LIN {X 0,Y 181.247,Z 724.094,A -85,B 0,C 180,E1 25006.197,E2 25006.197} C_VEL
LIN {X 0,Y 212.827,Z 697.919,A -85,B 0,C 180,E1 25010.796,E2 25010.796} C_VEL
LIN {X 0,Y 227.243,Z 683.519,A -85,B 0,C 180,E1 25012.44,E2 25012.44} C_VEL
LIN {X 0,Y 228.905,Z 680.992,A -85,B 0,C 180,E1 25016.21,E2 25016.21} C_VEL
LIN {X 0,Y 228.998,Z 681.06,A -85,B 0,C 180,E1 25020.002,E2 25020.002} C_VEL
LIN {X 0,Y 227.551,Z 683.584,A -85,B 0,C 180,E1 25023.524,E2 25023.524} C_VEL
LIN {X 0,Y 198.346,Z 711.493,A -85,B 0,C 180,E1 25027.069,E2 25027.069} C_VEL
LIN {X 0,Y 166.945,Z 735.496,A -85,B 0,C 180,E1 25032.577,E2 25032.577} C_VEL
LIN {X 0,Y 134.271,Z 755.47,A -85,B 0,C 180,E1 25041.514,E2 25041.514} C_VEL
LIN {X 0,Y 104.1,Z 770.587,A -85,B 0,C 180,E1 25057.124,E2 25057.124} C_VEL
LIN {X 0,Y 86.325,Z 778.801,A -85,B 0,C 180,E1 25078.251,E2 25078.251} C_VEL
LIN {X 0,Y 80.671,Z 781.977,A -85,B 0,C 180,E1 25099.182,E2 25099.182} C_VEL
LIN {X 0,Y 80.808,Z 782.413,A -85,B 0,C 180,E1 25110,E2 25110} C_VEL
LIN {X 0,Y 83.389,Z 780.22,A -85,B 0,C 180,E1 25134.788,E2 25134.788} C_VEL
LIN {X 0,Y 97.45,Z 773.708,A -85,B 0,C 180,E1 25157.173,E2 25157.173} C_VEL
LIN {X 0,Y 123.333,Z 761.326,A -85,B 0,C 180,E1 25174.086,E2 25174.086} C_VEL
LIN {X 0,Y 156.668,Z 742.373,A -85,B 0,C 180,E1 25185.118,E2 25185.118} C_VEL
LIN {X 0,Y 191.224,Z 717.631,A -85,B 0,C 180,E1 25191.795,E2 25191.795} C_VEL
LIN {X 0,Y 222.942,Z 688.687,A -85,B 0,C 180,E1 25195.995,E2 25195.995} C_VEL
LIN {X 0,Y 227.55,Z 683.825,A -85,B 0,C 180,E1 25196.478,E2 25196.478} C_VEL
LIN {X 0,Y 229.058,Z 681.251,A -85,B 0,C 180,E1 25199.998,E2 25199.998} C_VEL
LIN {X 0,Y 228.87,Z 681.291,A -85,B 0,C 180,E1 25203.791,E2 25203.791} C_VEL
LIN {X 0,Y 227.892,Z 682.996,A -85,B 0,C 180,E1 25207.158,E2 25207.158} C_VEL
LIN {X 0,Y 219.93,Z 691.3,A -85,B 0,C 180,E1 25208.319,E2 25208.319} C_VEL
LIN {X 0,Y 189.42,Z 718.093,A -85,B 0,C 180,E1 25212.372,E2 25212.372} C_VEL
LIN {X 0,Y 157.043,Z 740.418,A -85,B 0,C 180,E1 25218.724,E2 25218.724} C_VEL
LIN {X 0,Y 125.362,Z 757.593,A -85,B 0,C 180,E1 25228.881,E2 25228.881} C_VEL
LIN {X 0,Y 98.281,Z 769.456,A -85,B 0,C 180,E1 25246.11,E2 25246.11} C_VEL
LIN {X 0,Y 83.688,Z 775.171,A -85,B 0,C 180,E1 25268.786,E2 25268.786} C_VEL
LIN {X 0,Y 81.015,Z 776.528,A -85,B 0,C 180,E1 25290,E2 25290} C_VEL
LIN {X 0,Y 83.704,Z 775.133,A -85,B 0,C 180,E1 25311.21,E2 25311.21} C_VEL
LIN {X 0,Y 98.34,Z 769.389,A -85,B 0,C 180,E1 25333.857,E2 25333.857} C_VEL
LIN {X 0,Y 126.011,Z 757.227,A -85,B 0,C 180,E1 25351.281,E2 25351.281} C_VEL
LIN {X 0,Y 148.843,Z 745.136,A -85,B 0,C 180,E1 25359.119,E2 25359.119} C_VEL
LIN {X 0,Y 159.683,Z 738.038,A -85,B 0,C 180,E1 25363.519,E2 25363.519} C_VEL
LIN {X 0,Y 171.008,Z 730.237,A -85,B 0,C 180,E1 25367.284,E2 25367.284} C_VEL
LIN {X 0,Y 202.656,Z 706.253,A -85,B 0,C 180,E1 25371.877,E2 25371.877} C_VEL
LIN {X 0,Y 222.664,Z 687.627,A -85,B 0,C 180,E1 25374.254,E2 25374.254} C_VEL
LIN {X 0,Y 223.276,Z 686.711,A -85,B 0,C 180,E1 25376.114,E2 25376.114} C_VEL
LIN {X 0,Y 222.89,Z 687.51,A -85,B 0,C 180,E1 25381.189,E2 25381.189} C_VEL
LIN {X 0,Y 221.964,Z 688.666,A -85,B 0,C 180,E1 25381.969,E2 25381.969} C_VEL
LIN {X 0,Y 190.199,Z 717.114,A -85,B 0,C 180,E1 25385.675,E2 25385.675} C_VEL
LIN {X 0,Y 154.741,Z 741.948,A -85,B 0,C 180,E1 25391.903,E2 25391.903} C_VEL
LIN {X 0,Y 120.508,Z 760.698,A -85,B 0,C 180,E1 25402.146,E2 25402.146} C_VEL
LIN {X 0,Y 90.513,Z 773.971,A -85,B 0,C 180,E1 25420.57,E2 25420.57} C_VEL
LIN {X 0,Y 75.014,Z 780.476,A -85,B 0,C 180,E1 25446.19,E2 25446.19} C_VEL
LIN {X 0,Y 72.87,Z 782.124,A -85,B 0,C 180,E1 25470,E2 25470} C_VEL
LIN {X 0,Y 75.013,Z 780.5,A -85,B 0,C 180,E1 25493.809,E2 25493.809} C_VEL
LIN {X 0,Y 90.48,Z 774.015,A -85,B 0,C 180,E1 25519.441,E2 25519.441} C_VEL
LIN {X 0,Y 120.494,Z 760.781,A -85,B 0,C 180,E1 25537.852,E2 25537.852} C_VEL
LIN {X 0,Y 154.748,Z 742.066,A -85,B 0,C 180,E1 25548.084,E2 25548.084} C_VEL
LIN {X 0,Y 190.221,Z 717.304,A -85,B 0,C 180,E1 25554.259,E2 25554.259} C_VEL
LIN {X 0,Y 222.009,Z 688.863,A -85,B 0,C 180,E1 25558.04,E2 25558.04} C_VEL
LIN {X 0,Y 223.412,Z 686.977,A -85,B 0,C 180,E1 25559.998,E2 25559.998} C_VEL
LIN {X 0,Y 222.855,Z 687.56,A -85,B 0,C 180,E1 25565.044,E2 25565.044} C_VEL
LIN {X 0,Y 222.649,Z 687.908,A -85,B 0,C 180,E1 25565.739,E2 25565.739} C_VEL
LIN {X 0,Y 190.138,Z 716.678,A -85,B 0,C 180,E1 25569.637,E2 25569.637} C_VEL
LIN {X 0,Y 157.034,Z 739.31,A -85,B 0,C 180,E1 25575.376,E2 25575.376} C_VEL
LIN {X 0,Y 121.669,Z 757.885,A -85,B 0,C 180,E1 25585.551,E2 25585.551} C_VEL
LIN {X 0,Y 92.636,Z 769.747,A -85,B 0,C 180,E1 25602.649,E2 25602.649} C_VEL
LIN {X 0,Y 76.32,Z 775.46,A -85,B 0,C 180,E1 25626.623,E2 25626.623} C_VEL
LIN {X 0,Y 73.116,Z 776.815,A -85,B 0,C 180,E1 25650,E2 25650} C_VEL
LIN {X 0,Y 76.336,Z 775.423,A -85,B 0,C 180,E1 25673.372,E2 25673.372} C_VEL
LIN {X 0,Y 92.69,Z 769.681,A -85,B 0,C 180,E1 25697.316,E2 25697.316} C_VEL
LIN {X 0,Y 122.329,Z 757.522,A -85,B 0,C 180,E1 25714.606,E2 25714.606} C_VEL
LIN {X 0,Y 157.068,Z 739.149,A -85,B 0,C 180,E1 25724.581,E2 25724.581} C_VEL
LIN {X 0,Y 171.008,Z 730.237,A -85,B 0,C 180,E1 25727.284,E2 25727.284} C_VEL
LIN {X 0,Y 182.635,Z 721.723,A -85,B 0,C 180,E1 25730.535,E2 25730.535} C_VEL
LIN {X 0,Y 192.75,Z 713.822,A -85,B 0,C 180,E1 25733.112,E2 25733.112} C_VEL
LIN {X 0,Y 194.377,Z 712.525,A -85,B 0,C 180,E1 25733.326,E2 25733.326} C_VEL
LIN {X 0,Y 216.534,Z 693.283,A -85,B 0,C 180,E1 25735.643,E2 25735.643} C_VEL
LIN {X 0,Y 217.51,Z 692.345,A -85,B 0,C 180,E1 25736.011,E2 25736.011} C_VEL
LIN {X 0,Y 217.609,Z 692.411,A -85,B 0,C 180,E1 25740.002,E2 25740.002} C_VEL
LIN {X 0,Y 202.192,Z 706.448,A -85,B 0,C 180,E1 25741.753,E2 25741.753} C_VEL
LIN {X 0,Y 169.875,Z 731.007,A -85,B 0,C 180,E1 25745.966,E2 25745.966} C_VEL
LIN {X 0,Y 135.641,Z 751.45,A -85,B 0,C 180,E1 25752.902,E2 25752.902} C_VEL
LIN {X 0,Y 103.811,Z 766.412,A -85,B 0,C 180,E1 25764.273,E2 25764.273} C_VEL
LIN {X 0,Y 76.451,Z 776.915,A -85,B 0,C 180,E1 25786.117,E2 25786.117} C_VEL
LIN {X 0,Y 67.715,Z 780.182,A -85,B 0,C 180,E1 25803.435,E2 25803.435} C_VEL
LIN {X 0,Y 64.928,Z 781.835,A -85,B 0,C 180,E1 25830,E2 25830} C_VEL
LIN {X 0,Y 67.715,Z 780.207,A -85,B 0,C 180,E1 25856.564,E2 25856.564} C_VEL
LIN {X 0,Y 84.983,Z 773.851,A -85,B 0,C 180,E1 25883.298,E2 25883.298} C_VEL
LIN {X 0,Y 115.267,Z 761.512,A -85,B 0,C 180,E1 25900.71,E2 25900.71} C_VEL
LIN {X 0,Y 149.728,Z 743.767,A -85,B 0,C 180,E1 25910.392,E2 25910.392} C_VEL
LIN {X 0,Y 184.033,Z 721.156,A -85,B 0,C 180,E1 25916.015,E2 25916.015} C_VEL
LIN {X 0,Y 215.219,Z 694.933,A -85,B 0,C 180,E1 25919.546,E2 25919.546} C_VEL
LIN {X 0,Y 217.661,Z 692.593,A -85,B 0,C 180,E1 25919.998,E2 25919.998} C_VEL
LIN {X 0,Y 217.464,Z 692.627,A -85,B 0,C 180,E1 25923.99,E2 25923.99} C_VEL
LIN {X 0,Y 205.321,Z 703.66,A -85,B 0,C 180,E1 25925.406,E2 25925.406} C_VEL
LIN {X 0,Y 174.486,Z 727.337,A -85,B 0,C 180,E1 25929.217,E2 25929.217} C_VEL
LIN {X 0,Y 141.335,Z 747.205,A -85,B 0,C 180,E1 25935.383,E2 25935.383} C_VEL
LIN {X 0,Y 106.184,Z 763.204,A -85,B 0,C 180,E1 25947.029,E2 25947.029} C_VEL
LIN {X 0,Y 78.516,Z 772.86,A -85,B 0,C 180,E1 25967.55,E2 25967.55} C_VEL
LIN {X 0,Y 65.738,Z 776.783,A -85,B 0,C 180,E1 25996.684,E2 25996.684} C_VEL
LIN {X 0,Y 65.199,Z 777.103,A -85,B 0,C 180,E1 26010,E2 26010} C_VEL
LIN {X 0,Y 69.067,Z 775.715,A -85,B 0,C 180,E1 26036.006,E2 26036.006} C_VEL
LIN {X 0,Y 87.414,Z 769.976,A -85,B 0,C 180,E1 26061.212,E2 26061.212} C_VEL
LIN {X 0,Y 118.16,Z 758.2,A -85,B 0,C 180,E1 26077.791,E2 26077.791} C_VEL
LIN {X 0,Y 151.659,Z 741.427,A -85,B 0,C 180,E1 26086.761,E2 26086.761} C_VEL
LIN {X 0,Y 186.136,Z 718.9,A -85,B 0,C 180,E1 26092.315,E2 26092.315} C_VEL
LIN {X 0,Y 194.377,Z 712.525,A -85,B 0,C 180,E1 26093.326,E2 26093.326} C_VEL
LIN {X 0,Y 201.791,Z 706.345,A -85,B 0,C 180,E1 26095.31,E2 26095.31} C_VEL
LIN {X 0,Y 209.229,Z 699.942,A -85,B 0,C 180,E1 26097.168,E2 26097.168} C_VEL
LIN {X 0,Y 211.637,Z 697.732,A -85,B 0,C 180,E1 26097.44,E2 26097.44} C_VEL
LIN {X 0,Y 211.653,Z 697.751,A -85,B 0,C 180,E1 26098.428,E2 26098.428} C_VEL
LIN {X 0,Y 178.493,Z 724.38,A -85,B 0,C 180,E1 26101.989,E2 26101.989} C_VEL
LIN {X 0,Y 141.371,Z 747.345,A -85,B 0,C 180,E1 26107.816,E2 26107.816} C_VEL
LIN {X 0,Y 103.874,Z 764.915,A -85,B 0,C 180,E1 26118.651,E2 26118.651} C_VEL
LIN {X 0,Y 73.922,Z 775.651,A -85,B 0,C 180,E1 26137.918,E2 26137.918} C_VEL
LIN {X 0,Y 60.577,Z 779.887,A -85,B 0,C 180,E1 26160.006,E2 26160.006} C_VEL
LIN {X 0,Y 56.982,Z 781.546,A -85,B 0,C 180,E1 26190,E2 26190} C_VEL
LIN {X 0,Y 60.577,Z 779.912,A -85,B 0,C 180,E1 26219.993,E2 26219.993} C_VEL
LIN {X 0,Y 80.339,Z 773.554,A -85,B 0,C 180,E1 26248.005,E2 26248.005} C_VEL
LIN {X 0,Y 113.917,Z 760.742,A -85,B 0,C 180,E1 26265.067,E2 26265.067} C_VEL
LIN {X 0,Y 152.199,Z 741.452,A -85,B 0,C 180,E1 26274.177,E2 26274.177} C_VEL
LIN {X 0,Y 189.004,Z 716.866,A -85,B 0,C 180,E1 26279.219,E2 26279.219} C_VEL
LIN {X 0,Y 211.675,Z 697.966,A -85,B 0,C 180,E1 26281.567,E2 26281.567} C_VEL
LIN {X 0,Y 211.631,Z 697.976,A -85,B 0,C 180,E1 26282.389,E2 26282.389} C_VEL
LIN {X 0,Y 178.862,Z 723.925,A -85,B 0,C 180,E1 26285.911,E2 26285.911} C_VEL
LIN {X 0,Y 142.918,Z 745.686,A -85,B 0,C 180,E1 26291.483,E2 26291.483} C_VEL
LIN {X 0,Y 108.803,Z 761.195,A -85,B 0,C 180,E1 26300.634,E2 26300.634} C_VEL
LIN {X 0,Y 77.457,Z 771.827,A -85,B 0,C 180,E1 26318.563,E2 26318.563} C_VEL
LIN {X 0,Y 61.971,Z 776.04,A -85,B 0,C 180,E1 26340.748,E2 26340.748} C_VEL
LIN {X 0,Y 57.308,Z 777.39,A -85,B 0,C 180,E1 26370,E2 26370} C_VEL
LIN {X 0,Y 61.987,Z 776.006,A -85,B 0,C 180,E1 26399.244,E2 26399.244} C_VEL
LIN {X 0,Y 81.872,Z 770.477,A -85,B 0,C 180,E1 26425.035,E2 26425.035} C_VEL
LIN {X 0,Y 115.675,Z 758.364,A -85,B 0,C 180,E1 26441.622,E2 26441.622} C_VEL
LIN {X 0,Y 153.563,Z 739.765,A -85,B 0,C 180,E1 26450.404,E2 26450.404} C_VEL
LIN {X 0,Y 188.557,Z 716.78,A -85,B 0,C 180,E1 26455.148,E2 26455.148} C_VEL
LIN {X 0,Y 209.229,Z 699.942,A -85,B 0,C 180,E1 26457.168,E2 26457.168} C_VEL
LIN {X 0,Y 204.922,Z 703.641,A -85,B 0,C 180,E1 26457.807,E2 26457.807} C_VEL
LIN {X 0,Y 181.831,Z 721.615,A -85,B 0,C 180,E1 26458.985,E2 26458.985} C_VEL
LIN {X 0,Y 145.944,Z 744.078,A -85,B 0,C 180,E1 26463.574,E2 26463.574} C_VEL
LIN {X 0,Y 108.338,Z 761.854,A -85,B 0,C 180,E1 26471.952,E2 26471.952} C_VEL
LIN {X 0,Y 76.315,Z 773.21,A -85,B 0,C 180,E1 26486.769,E2 26486.769} C_VEL
LIN {X 0,Y 53.706,Z 779.591,A -85,B 0,C 180,E1 26515.677,E2 26515.677} C_VEL
LIN {X 0,Y 49.033,Z 781.257,A -85,B 0,C 180,E1 26550,E2 26550} C_VEL
LIN {X 0,Y 53.706,Z 779.617,A -85,B 0,C 180,E1 26584.323,E2 26584.323} C_VEL
LIN {X 0,Y 76.3,Z 773.256,A -85,B 0,C 180,E1 26613.252,E2 26613.252} C_VEL
LIN {X 0,Y 111.793,Z 760.549,A -85,B 0,C 180,E1 26629.097,E2 26629.097} C_VEL
LIN {X 0,Y 151.583,Z 741.144,A -85,B 0,C 180,E1 26637.284,E2 26637.284} C_VEL
LIN {X 0,Y 188.507,Z 716.976,A -85,B 0,C 180,E1 26641.669,E2 26641.669} C_VEL
LIN {X 0,Y 191.373,Z 714.748,A -85,B 0,C 180,E1 26642.024,E2 26642.024} C_VEL
LIN {X 0,Y 156.477,Z 737.848,A -85,B 0,C 180,E1 26645.961,E2 26645.961} C_VEL
LIN {X 0,Y 120.248,Z 755.874,A -85,B 0,C 180,E1 26652.614,E2 26652.614} C_VEL
LIN {X 0,Y 84.15,Z 768.892,A -85,B 0,C 180,E1 26665.887,E2 26665.887} C_VEL
LIN {X 0,Y 56.791,Z 775.921,A -85,B 0,C 180,E1 26693.092,E2 26693.092} C_VEL
LIN {X 0,Y 49.387,Z 777.678,A -85,B 0,C 180,E1 26730,E2 26730} C_VEL
LIN {X 0,Y 56.831,Z 775.882,A -85,B 0,C 180,E1 26766.961,E2 26766.961} C_VEL
LIN {X 0,Y 84.193,Z 768.822,A -85,B 0,C 180,E1 26794.054,E2 26794.054} C_VEL
LIN {X 0,Y 116.814,Z 757.258,A -85,B 0,C 180,E1 26806.446,E2 26806.446} C_VEL
LIN {X 0,Y 154.648,Z 738.775,A -85,B 0,C 180,E1 26813.713,E2 26813.713} C_VEL
LIN {X 0,Y 189.551,Z 715.947,A -85,B 0,C 180,E1 26817.719,E2 26817.719} C_VEL
LIN {X 0,Y 191.985,Z 714.078,A -85,B 0,C 180,E1 26817.933,E2 26817.933} C_VEL
LIN {X 0,Y 181.831,Z 721.615,A -85,B 0,C 180,E1 26818.985,E2 26818.985} C_VEL
LIN {X 0,Y 172.823,Z 727.819,A -85,B 0,C 180,E1 26819.184,E2 26819.184} C_VEL
LIN {X 0,Y 152.331,Z 740.022,A -85,B 0,C 180,E1 26816.496,E2 26816.496} C_VEL
LIN {X 0,Y 115.188,Z 757.557,A -85,B 0,C 180,E1 26810.357,E2 26810.357} C_VEL
LIN {X 0,Y 80.983,Z 769.118,A -85,B 0,C 180,E1 26799.204,E2 26799.204} C_VEL
LIN {X 0,Y 57.584,Z 774.837,A -85,B 0,C 180,E1 26782.077,E2 26782.077} C_VEL
LIN {X 0,Y 42.9,Z 777.63,A -85,B 0,C 180,E1 26750.668,E2 26750.668} C_VEL
LIN {X 0,Y 41.464,Z 777.966,A -85,B 0,C 180,E1 26730,E2 26730} C_VEL
LIN {X 0,Y 48.652,Z 776.621,A -85,B 0,C 180,E1 26691.506,E2 26691.506} C_VEL
LIN {X 0,Y 75.339,Z 770.743,A -85,B 0,C 180,E1 26663.69,E2 26663.69} C_VEL
LIN {X 0,Y 111.601,Z 759.053,A -85,B 0,C 180,E1 26650.381,E2 26650.381} C_VEL
LIN {X 0,Y 151.7,Z 740.526,A -85,B 0,C 180,E1 26643.523,E2 26643.523} C_VEL
LIN {X 0,Y 162.247,Z 734.495,A -85,B 0,C 180,E1 26642.292,E2 26642.292} C_VEL
LIN {X 0,Y 155.216,Z 738.62,A -85,B 0,C 180,E1 26640.857,E2 26640.857} C_VEL
LIN {X 0,Y 117.805,Z 757.219,A -85,B 0,C 180,E1 26634.934,E2 26634.934} C_VEL
LIN {X 0,Y 79.362,Z 771.092,A -85,B 0,C 180,E1 26622.543,E2 26622.543} C_VEL
LIN {X 0,Y 55.913,Z 777.351,A -85,B 0,C 180,E1 26604.331,E2 26604.331} C_VEL
LIN {X 0,Y 41.993,Z 780.533,A -85,B 0,C 180,E1 26571.134,E2 26571.134} C_VEL
LIN {X 0,Y 41.081,Z 780.968,A -85,B 0,C 180,E1 26550,E2 26550} C_VEL
LIN {X 0,Y 47.226,Z 779.296,A -85,B 0,C 180,E1 26510.116,E2 26510.116} C_VEL
LIN {X 0,Y 72.975,Z 772.911,A -85,B 0,C 180,E1 26480.983,E2 26480.983} C_VEL
LIN {X 0,Y 110.525,Z 760.163,A -85,B 0,C 180,E1 26466.678,E2 26466.678} C_VEL
LIN {X 0,Y 151.417,Z 740.7,A -85,B 0,C 180,E1 26459.607,E2 26459.607} C_VEL
LIN {X 0,Y 161.204,Z 734.991,A -85,B 0,C 180,E1 26458.425,E2 26458.425} C_VEL
LIN {X 0,Y 162.781,Z 734.044,A -85,B 0,C 180,E1 26457.68,E2 26457.68} C_VEL
LIN {X 0,Y 152.331,Z 740.022,A -85,B 0,C 180,E1 26456.496,E2 26456.496} C_VEL
LIN {X 0,Y 136.8,Z 748.109,A -85,B 0,C 180,E1 26456.064,E2 26456.064} C_VEL
LIN {X 0,Y 120.79,Z 755.142,A -85,B 0,C 180,E1 26455.486,E2 26455.486} C_VEL
LIN {X 0,Y 85.388,Z 767.551,A -85,B 0,C 180,E1 26447.236,E2 26447.236} C_VEL
LIN {X 0,Y 53.031,Z 775.13,A -85,B 0,C 180,E1 26428.933,E2 26428.933} C_VEL
LIN {X 0,Y 35.561,Z 777.92,A -85,B 0,C 180,E1 26395.201,E2 26395.201} C_VEL
LIN {X 0,Y 33.54,Z 778.254,A -85,B 0,C 180,E1 26370.001,E2 26370.001} C_VEL
LIN {X 0,Y 42.693,Z 776.911,A -85,B 0,C 180,E1 26324.821,E2 26324.821} C_VEL
LIN {X 0,Y 72.473,Z 771.035,A -85,B 0,C 180,E1 26297.834,E2 26297.834} C_VEL
LIN {X 0,Y 110.43,Z 759.348,A -85,B 0,C 180,E1 26286.246,E2 26286.246} C_VEL
LIN {X 0,Y 136.372,Z 748.386,A -85,B 0,C 180,E1 26282.198,E2 26282.198} C_VEL
LIN {X 0,Y 136.338,Z 748.421,A -85,B 0,C 180,E1 26281.788,E2 26281.788} C_VEL
LIN {X 0,Y 96.842,Z 764.718,A -85,B 0,C 180,E1 26274.678,E2 26274.678} C_VEL
LIN {X 0,Y 58.147,Z 775.626,A -85,B 0,C 180,E1 26257.693,E2 26257.693} C_VEL
LIN {X 0,Y 34.612,Z 780.24,A -85,B 0,C 180,E1 26215.941,E2 26215.941} C_VEL
LIN {X 0,Y 33.123,Z 780.679,A -85,B 0,C 180,E1 26189.999,E2 26189.999} C_VEL
LIN {X 0,Y 41.327,Z 779,A -85,B 0,C 180,E1 26142.882,E2 26142.882} C_VEL
LIN {X 0,Y 70.443,Z 772.612,A -85,B 0,C 180,E1 26114.701,E2 26114.701} C_VEL
LIN {X 0,Y 109.87,Z 759.861,A -85,B 0,C 180,E1 26102.383,E2 26102.383} C_VEL
LIN {X 0,Y 136.341,Z 748.307,A -85,B 0,C 180,E1 26098.189,E2 26098.189} C_VEL
LIN {X 0,Y 136.381,Z 748.265,A -85,B 0,C 180,E1 26097.71,E2 26097.71} C_VEL
LIN {X 0,Y 120.79,Z 755.142,A -85,B 0,C 180,E1 26095.486,E2 26095.486} C_VEL
LIN {X 0,Y 104.432,Z 761.387,A -85,B 0,C 180,E1 26094.689,E2 26094.689} C_VEL
LIN {X 0,Y 87.842,Z 766.728,A -85,B 0,C 180,E1 26093.6,E2 26093.6} C_VEL
LIN {X 0,Y 49.364,Z 775.423,A -85,B 0,C 180,E1 26076.955,E2 26076.955} C_VEL
LIN {X 0,Y 28.559,Z 778.21,A -85,B 0,C 180,E1 26042.018,E2 26042.018} C_VEL
LIN {X 0,Y 25.632,Z 778.542,A -85,B 0,C 180,E1 26010.001,E2 26010.001} C_VEL
LIN {X 0,Y 37.476,Z 777.203,A -85,B 0,C 180,E1 25956.095,E2 25956.095} C_VEL
LIN {X 0,Y 70.902,Z 771.225,A -85,B 0,C 180,E1 25931.383,E2 25931.383} C_VEL
LIN {X 0,Y 109.889,Z 759.633,A -85,B 0,C 180,E1 25921.923,E2 25921.923} C_VEL
LIN {X 0,Y 68.811,Z 772.362,A -85,B 0,C 180,E1 25911.968,E2 25911.968} C_VEL
LIN {X 0,Y 36.285,Z 778.732,A -85,B 0,C 180,E1 25886.571,E2 25886.571} C_VEL
LIN {X 0,Y 25.171,Z 780.389,A -85,B 0,C 180,E1 25829.999,E2 25829.999} C_VEL
LIN {X 0,Y 36.285,Z 778.704,A -85,B 0,C 180,E1 25773.428,E2 25773.428} C_VEL
LIN {X 0,Y 68.814,Z 772.313,A -85,B 0,C 180,E1 25748.046,E2 25748.046} C_VEL
LIN {X 0,Y 110.102,Z 759.464,A -85,B 0,C 180,E1 25738.03,E2 25738.03} C_VEL
LIN {X 0,Y 87.842,Z 766.728,A -85,B 0,C 180,E1 25733.6,E2 25733.6} C_VEL
LIN {X 0,Y 70.983,Z 771.159,A -85,B 0,C 180,E1 25732.064,E2 25732.064} C_VEL
LIN {X 0,Y 53.947,Z 774.55,A -85,B 0,C 180,E1 25729.643,E2 25729.643} C_VEL
LIN {X 0,Y 22.208,Z 778.5,A -85,B 0,C 180,E1 25692.985,E2 25692.985} C_VEL
LIN {X 0,Y 17.703,Z 778.83,A -85,B 0,C 180,E1 25650.001,E2 25650.001} C_VEL
LIN {X 0,Y 33.399,Z 777.493,A -85,B 0,C 180,E1 25584.949,E2 25584.949} C_VEL
LIN {X 0,Y 71.852,Z 771.064,A -85,B 0,C 180,E1 25564.299,E2 25564.299} C_VEL
LIN {X 0,Y 81.32,Z 768.714,A -85,B 0,C 180,E1 25561.899,E2 25561.899} C_VEL
LIN {X 0,Y 46.128,Z 776.459,A -85,B 0,C 180,E1 25549.974,E2 25549.974} C_VEL
LIN {X 0,Y 21.055,Z 779.691,A -85,B 0,C 180,E1 25513.99,E2 25513.99} C_VEL
LIN {X 0,Y 17.203,Z 780.1,A -85,B 0,C 180,E1 25469.999,E2 25469.999} C_VEL
LIN {X 0,Y 32.529,Z 778.409,A -85,B 0,C 180,E1 25401.415,E2 25401.415} C_VEL
LIN {X 0,Y 72.576,Z 770.962,A -85,B 0,C 180,E1 25380.007,E2 25380.007} C_VEL
LIN {X 0,Y 81.58,Z 768.582,A -85,B 0,C 180,E1 25378.068,E2 25378.068} C_VEL
LIN {X 0,Y 53.947,Z 774.55,A -85,B 0,C 180,E1 25369.643,E2 25369.643} C_VEL
LIN {X 0,Y 41.24,Z 776.509,A -85,B 0,C 180,E1 25366.335,E2 25366.335} C_VEL
LIN {X 0,Y 21.744,Z 778.458,A -85,B 0,C 180,E1 25359.462,E2 25359.462} C_VEL
LIN {X 0,Y 19.8,Z 778.582,A -85,B 0,C 180,E1 25356.606,E2 25356.606} C_VEL
LIN {X 0,Y 9.794,Z 779.118,A -85,B 0,C 180,E1 25290.002,E2 25290.002} C_VEL
LIN {X 0,Y 30.884,Z 777.785,A -85,B 0,C 180,E1 25211.325,E2 25211.325} C_VEL
LIN {X 0,Y 50.751,Z 775.26,A -85,B 0,C 180,E1 25201.893,E2 25201.893} C_VEL
LIN {X 0,Y 16.676,Z 779.363,A -85,B 0,C 180,E1 25175.228,E2 25175.228} C_VEL
LIN {X 0,Y 9.231,Z 779.81,A -85,B 0,C 180,E1 25109.998,E2 25109.998} C_VEL
LIN {X 0,Y 30.511,Z 778.112,A -85,B 0,C 180,E1 25027.016,E2 25027.016} C_VEL
LIN {X 0,Y 50.833,Z 775.205,A -85,B 0,C 180,E1 25018.089,E2 25018.089} C_VEL
LIN {X 0,Y 19.8,Z 778.582,A -85,B 0,C 180,E1 24996.606,E2 24996.606} C_VEL
LIN {X 0,Y 11.606,Z 779.087,A -85,B 0,C 180,E1 24985.498,E2 24985.498} C_VEL
LIN {X 0,Y 4.548,Z 779.346,A -85,B 0,C 180,E1 24851.236,E2 24851.236} C_VEL
LIN {X 0,Y 8.548,Z 779.291,A -85,B 0,C 180,E1 24839.943,E2 24839.943} C_VEL
LIN {X 0,Y 1.249,Z 779.52,A -85,B 0,C 180,E1 24749.986,E2 24749.986} C_VEL
LIN {X 0,Y 8.502,Z 779.287,A -85,B 0,C 180,E1 24660.057,E2 24660.057} C_VEL
LIN {X 0,Y 1.863,Z 779.406,A -85,B 0,C 180,E1 24570.01,E2 24570.01} C_VEL
LIN {X 0,Y 4.548,Z 779.346,A -85,B 0,C 180,E1 24491.236,E2 24491.236} C_VEL
LIN {X 0,Y 6.456,Z 781.346,A -85,B 0,C 180,E1 24484.022,E2 24484.022} C_VEL
LIN {X 0,Y 6.456,Z 799,A -85,B 0,C 180,E1 24484.022,E2 24484.022} C_VEL
LIN {X 0,Y 6.456,Z 799,A -85,B 0,C 180,E1 24484.022,E2 24484.022}

QRS_NEXT_CUT()
PTP {E1 24656.919,E2 24656.919}
PTP {X 0,Y 607.906,A -85,B 0,C 180,E1 24656.919,E2 24656.919,E3 0,E4 0,E5 0,E6 0}
QRS_SPEED_INIT()
LIN {X 0,Y 607.906,Z 799,A -85,B 0,C 180,E1 24656.919,E2 24656.919,E3 0,E4 0,E5 0,E6 0} C_VEL
LIN {X 0,Y 607.906,Z 136.404,A -85,B 0,C 180,E1 24656.919,E2 24656.919} C_VEL
LIN {X 0,Y 607.906,Z 128.326,A -85,B 0,C 180,E1 24656.919,E2 24656.919} C_VEL
LIN {X 0,Y 607.886,Z 126.326,A -85,B 0,C 180,E1 24656.73,E2 24656.73} C_VEL
LIN {X 0,Y 607.894,Z 126.321,A -85,B 0,C 180,E1 24653.673,E2 24653.673} C_VEL
LIN {X 0,Y 607.867,Z 126.325,A -85,B 0,C 180,E1 24650.532,E2 24650.532} C_VEL
LIN {X 0,Y 607.914,Z 126.321,A -85,B 0,C 180,E1 24647.461,E2 24647.461} C_VEL
LIN {X 0,Y 607.856,Z 126.325,A -85,B 0,C 180,E1 24644.35,E2 24644.35} C_VEL
LIN {X 0,Y 607.918,Z 126.323,A -85,B 0,C 180,E1 24641.293,E2 24641.293} C_VEL
LIN {X 0,Y 607.849,Z 126.325,A -85,B 0,C 180,E1 24638.278,E2 24638.278} C_VEL
LIN {X 0,Y 607.914,Z 126.326,A -85,B 0,C 180,E1 24635.203,E2 24635.203} C_VEL
LIN {X 0,Y 607.845,Z 126.325,A -85,B 0,C 180,E1 24632.15,E2 24632.15} C_VEL
LIN {X 0,Y 607.912,Z 126.327,A -85,B 0,C 180,E1 24629.125,E2 24629.125} C_VEL
LIN {X 0,Y 607.84,Z 126.326,A -85,B 0,C 180,E1 24626.108,E2 24626.108} C_VEL
LIN {X 0,Y 607.885,Z 126.327,A -85,B 0,C 180,E1 24622.986,E2 24622.986} C_VEL
LIN {X 0,Y 607.835,Z 126.326,A -85,B 0,C 180,E1 24620.094,E2 24620.094} C_VEL
LIN {X 0,Y 607.888,Z 126.327,A -85,B 0,C 180,E1 24617.047,E2 24617.047} C_VEL
LIN {X 0,Y 607.829,Z 126.328,A -85,B 0,C 180,E1 24614.176,E2 24614.176} C_VEL
LIN {X 0,Y 607.901,Z 126.327,A -85,B 0,C 180,E1 24611.122,E2 24611.122} C_VEL
LIN {X 0,Y 607.835,Z 126.321,A -85,B 0,C 180,E1 24608.16,E2 24608.16} C_VEL
LIN {X 0,Y 607.884,Z 126.625,A -85,B 0,C 180,E1 24607.518,E2 24607.518} C_VEL
LIN {X 0,Y 607.917,Z 133.876,A -85,B 0,C 180,E1 24607.01,E2 24607.01} C_VEL
LIN {X 0,Y 607.883,Z 179.67,A -85,B 0,C 180,E1 24604.116,E2 24604.116} C_VEL
LIN {X 0,Y 607.91,Z 208.953,A -85,B 0,C 180,E1 24602.326,E2 24602.326} C_VEL
LIN {X 0,Y 607.917,Z 431.782,A -85,B 0,C 180,E1 24599.317,E2 24599.317} C_VEL
LIN {X 0,Y 607.901,Z 514.758,A -85,B 0,C 180,E1 24598.193,E2 24598.193} C_VEL
LIN {X 0,Y 607.907,Z 535.55,A -85,B 0,C 180,E1 24597.739,E2 24597.739} C_VEL
LIN {X 0,Y 607.914,Z 556.34,A -85,B 0,C 180,E1 24597.127,E2 24597.127} C_VEL
LIN {X 0,Y 607.914,Z 576.273,A -85,B 0,C 180,E1 24596.364,E2 24596.364} C_VEL
LIN {X 0,Y 607.919,Z 597.393,A -85,B 0,C 180,E1 24595.368,E2 24595.368} C_VEL
LIN {X 0,Y 607.917,Z 616.727,A -85,B 0,C 180,E1 24594.278,E2 24594.278} C_VEL
LIN {X 0,Y 607.915,Z 635.158,A -85,B 0,C 180,E1 24593.044,E2 24593.044} C_VEL
LIN {X 0,Y 607.91,Z 652.748,A -85,B 0,C 180,E1 24591.677,E2 24591.677} C_VEL
LIN {X 0,Y 607.914,Z 669.702,A -85,B 0,C 180,E1 24590.155,E2 24590.155} C_VEL
LIN {X 0,Y 607.917,Z 685.582,A -85,B 0,C 180,E1 24588.507,E2 24588.507} C_VEL
LIN {X 0,Y 607.914,Z 700.26,A -85,B 0,C 180,E1 24586.728,E2 24586.728} C_VEL
LIN {X 0,Y 607.914,Z 712.749,A -85,B 0,C 180,E1 24584.964,E2 24584.964} C_VEL
LIN {X 0,Y 607.914,Z 723.99,A -85,B 0,C 180,E1 24583.119,E2 24583.119} C_VEL
LIN {X 0,Y 607.903,Z 733.345,A -85,B 0,C 180,E1 24581.287,E2 24581.287} C_VEL
LIN {X 0,Y 607.903,Z 741.797,A -85,B 0,C 180,E1 24579.276,E2 24579.276} C_VEL
LIN {X 0,Y 607.904,Z 748.508,A -85,B 0,C 180,E1 24577.276,E2 24577.276} C_VEL
LIN {X 0,Y 607.905,Z 753.211,A -85,B 0,C 180,E1 24575.379,E2 24575.379} C_VEL
LIN {X 0,Y 607.918,Z 756.791,A -85,B 0,C 180,E1 24573.291,E2 24573.291} C_VEL
LIN {X 0,Y 607.908,Z 758.682,A -85,B 0,C 180,E1 24571.225,E2 24571.225} C_VEL
LIN {X 0,Y 607.903,Z 758.839,A -85,B 0,C 180,E1 24569.246,E2 24569.246} C_VEL
LIN {X 0,Y 607.912,Z 757.336,A -85,B 0,C 180,E1 24567.077,E2 24567.077} C_VEL
LIN {X 0,Y 607.909,Z 754.403,A -85,B 0,C 180,E1 24565.094,E2 24565.094} C_VEL
LIN {X 0,Y 607.91,Z 749.765,A -85,B 0,C 180,E1 24563.104,E2 24563.104} C_VEL
LIN {X 0,Y 607.918,Z 743.196,A -85,B 0,C 180,E1 24561.011,E2 24561.011} C_VEL
LIN {X 0,Y 607.908,Z 735.493,A -85,B 0,C 180,E1 24559.088,E2 24559.088} C_VEL
LIN {X 0,Y 607.904,Z 726.031,A -85,B 0,C 180,E1 24557.171,E2 24557.171} C_VEL
LIN {X 0,Y 607.902,Z 714.872,A -85,B 0,C 180,E1 24555.268,E2 24555.268} C_VEL
LIN {X 0,Y 607.904,Z 702.446,A -85,B 0,C 180,E1 24553.469,E2 24553.469} C_VEL
LIN {X 0,Y 607.915,Z 688.905,A -85,B 0,C 180,E1 24551.791,E2 24551.791} C_VEL
LIN {X 0,Y 607.913,Z 672.636,A -85,B 0,C 180,E1 24550.046,E2 24550.046} C_VEL
LIN {X 0,Y 607.917,Z 655.729,A -85,B 0,C 180,E1 24548.484,E2 24548.484} C_VEL
LIN {X 0,Y 607.914,Z 637.883,A -85,B 0,C 180,E1 24547.058,E2 24547.058} C_VEL
LIN {X 0,Y 607.917,Z 618.932,A -85,B 0,C 180,E1 24545.773,E2 24545.773} C_VEL
LIN {X 0,Y 607.919,Z 599.109,A -85,B 0,C 180,E1 24544.632,E2 24544.632} C_VEL
LIN {X 0,Y 607.914,Z 579.672,A -85,B 0,C 180,E1 24543.687,E2 24543.687} C_VEL
LIN {X 0,Y 607.916,Z 559.525,A -85,B 0,C 180,E1 24542.898,E2 24542.898} C_VEL
LIN {X 0,Y 607.91,Z 537.299,A -85,B 0,C 180,E1 24542.215,E2 24542.215} C_VEL
LIN {X 0,Y 607.9,Z 516.862,A -85,B 0,C 180,E1 24541.753,E2 24541.753} C_VEL
LIN {X 0,Y 607.913,Z 477.868,A -85,B 0,C 180,E1 24541.203,E2 24541.203} C_VEL
LIN {X 0,Y 607.884,Z 248.819,A -85,B 0,C 180,E1 24538.132,E2 24538.132} C_VEL
LIN {X 0,Y 607.917,Z 208.712,A -85,B 0,C 180,E1 24537.577,E2 24537.577} C_VEL
LIN {X 0,Y 607.917,Z 160.031,A -85,B 0,C 180,E1 24534.567,E2 24534.567} C_VEL
LIN {X 0,Y 607.89,Z 126.798,A -85,B 0,C 180,E1 24532.421,E2 24532.421} C_VEL
LIN {X 0,Y 607.86,Z 126.32,A -85,B 0,C 180,E1 24532.143,E2 24532.143} C_VEL
LIN {X 0,Y 607.853,Z 126.326,A -85,B 0,C 180,E1 24529.315,E2 24529.315} C_VEL
LIN {X 0,Y 607.846,Z 126.327,A -85,B 0,C 180,E1 24526.042,E2 24526.042} C_VEL
LIN {X 0,Y 607.855,Z 126.326,A -85,B 0,C 180,E1 24523.225,E2 24523.225} C_VEL
LIN {X 0,Y 607.838,Z 126.327,A -85,B 0,C 180,E1 24520.029,E2 24520.029} C_VEL
LIN {X 0,Y 607.849,Z 126.328,A -85,B 0,C 180,E1 24517.239,E2 24517.239} C_VEL
LIN {X 0,Y 607.839,Z 126.327,A -85,B 0,C 180,E1 24514.001,E2 24514.001} C_VEL
LIN {X 0,Y 607.858,Z 126.327,A -85,B 0,C 180,E1 24511.205,E2 24511.205} C_VEL
LIN {X 0,Y 607.849,Z 126.326,A -85,B 0,C 180,E1 24508.063,E2 24508.063} C_VEL
LIN {X 0,Y 607.864,Z 126.326,A -85,B 0,C 180,E1 24505.215,E2 24505.215} C_VEL
LIN {X 0,Y 607.852,Z 126.325,A -85,B 0,C 180,E1 24502.027,E2 24502.027} C_VEL
LIN {X 0,Y 607.882,Z 126.326,A -85,B 0,C 180,E1 24499.106,E2 24499.106} C_VEL
LIN {X 0,Y 607.854,Z 126.324,A -85,B 0,C 180,E1 24495.944,E2 24495.944} C_VEL
LIN {X 0,Y 607.909,Z 126.327,A -85,B 0,C 180,E1 24492.926,E2 24492.926} C_VEL
LIN {X 0,Y 607.857,Z 126.324,A -85,B 0,C 180,E1 24489.849,E2 24489.849} C_VEL
LIN {X 0,Y 607.917,Z 126.325,A -85,B 0,C 180,E1 24486.801,E2 24486.801} C_VEL
LIN {X 0,Y 607.861,Z 126.324,A -85,B 0,C 180,E1 24483.678,E2 24483.678} C_VEL
LIN {X 0,Y 607.918,Z 126.32,A -85,B 0,C 180,E1 24480.566,E2 24480.566} C_VEL
LIN {X 0,Y 607.873,Z 126.325,A -85,B 0,C 180,E1 24477.455,E2 24477.455} C_VEL
LIN {X 0,Y 607.894,Z 126.32,A -85,B 0,C 180,E1 24474.242,E2 24474.242} C_VEL
LIN {X 0,Y 607.908,Z 126.327,A -85,B 0,C 180,E1 24471.106,E2 24471.106} C_VEL
LIN {X 0,Y 607.878,Z 126.321,A -85,B 0,C 180,E1 24467.943,E2 24467.943} C_VEL
LIN {X 0,Y 607.912,Z 126.323,A -85,B 0,C 180,E1 24464.84,E2 24464.84} C_VEL
LIN {X 0,Y 607.879,Z 126.323,A -85,B 0,C 180,E1 24461.69,E2 24461.69} C_VEL
LIN {X 0,Y 607.911,Z 126.319,A -85,B 0,C 180,E1 24458.575,E2 24458.575} C_VEL
LIN {X 0,Y 607.892,Z 126.325,A -85,B 0,C 180,E1 24455.409,E2 24455.409} C_VEL
LIN {X 0,Y 607.902,Z 126.318,A -85,B 0,C 180,E1 24452.153,E2 24452.153} C_VEL
LIN {X 0,Y 607.909,Z 126.324,A -85,B 0,C 180,E1 24448.969,E2 24448.969} C_VEL
LIN {X 0,Y 607.89,Z 126.321,A -85,B 0,C 180,E1 24445.823,E2 24445.823} C_VEL
LIN {X 0,Y 607.901,Z 126.322,A -85,B 0,C 180,E1 24442.752,E2 24442.752} C_VEL
LIN {X 0,Y 607.895,Z 126.323,A -85,B 0,C 180,E1 24439.598,E2 24439.598} C_VEL
LIN {X 0,Y 607.91,Z 126.317,A -85,B 0,C 180,E1 24436.358,E2 24436.358} C_VEL
LIN {X 0,Y 607.905,Z 126.323,A -85,B 0,C 180,E1 24433.044,E2 24433.044} C_VEL
LIN {X 0,Y 607.899,Z 126.31,A -85,B 0,C 180,E1 24429.816,E2 24429.816} C_VEL
LIN {X 0,Y 607.902,Z 126.639,A -85,B 0,C 180,E1 24429.521,E2 24429.521} C_VEL
LIN {X 0,Y 607.919,Z 130.809,A -85,B 0,C 180,E1 24429.226,E2 24429.226} C_VEL
LIN {X 0,Y 607.917,Z 161.328,A -85,B 0,C 180,E1 24427.383,E2 24427.383} C_VEL
LIN {X 0,Y 607.919,Z 357.497,A -85,B 0,C 180,E1 24424.57,E2 24424.57} C_VEL
LIN {X 0,Y 607.914,Z 509.002,A -85,B 0,C 180,E1 24422.443,E2 24422.443} C_VEL
LIN {X 0,Y 607.915,Z 532.149,A -85,B 0,C 180,E1 24421.955,E2 24421.955} C_VEL
LIN {X 0,Y 607.918,Z 551.554,A -85,B 0,C 180,E1 24421.394,E2 24421.394} C_VEL
LIN {X 0,Y 607.912,Z 572.95,A -85,B 0,C 180,E1 24420.627,E2 24420.627} C_VEL
LIN {X 0,Y 607.919,Z 593.115,A -85,B 0,C 180,E1 24419.725,E2 24419.725} C_VEL
LIN {X 0,Y 607.916,Z 613.778,A -85,B 0,C 180,E1 24418.648,E2 24418.648} C_VEL
LIN {X 0,Y 607.918,Z 633.576,A -85,B 0,C 180,E1 24417.42,E2 24417.42} C_VEL
LIN {X 0,Y 607.914,Z 652.968,A -85,B 0,C 180,E1 24416.049,E2 24416.049} C_VEL
LIN {X 0,Y 607.91,Z 671.187,A -85,B 0,C 180,E1 24414.558,E2 24414.558} C_VEL
LIN {X 0,Y 607.904,Z 689.604,A -85,B 0,C 180,E1 24412.84,E2 24412.84} C_VEL
LIN {X 0,Y 607.92,Z 705.881,A -85,B 0,C 180,E1 24411.111,E2 24411.111} C_VEL
LIN {X 0,Y 607.918,Z 721.059,A -85,B 0,C 180,E1 24409.253,E2 24409.253} C_VEL
LIN {X 0,Y 607.918,Z 735.52,A -85,B 0,C 180,E1 24407.22,E2 24407.22} C_VEL
LIN {X 0,Y 607.9,Z 747.037,A -85,B 0,C 180,E1 24405.355,E2 24405.355} C_VEL
LIN {X 0,Y 607.906,Z 757.756,A -85,B 0,C 180,E1 24403.312,E2 24403.312} C_VEL
LIN {X 0,Y 607.915,Z 766.785,A -85,B 0,C 180,E1 24401.287,E2 24401.287} C_VEL
LIN {X 0,Y 607.908,Z 774.343,A -85,B 0,C 180,E1 24399.18,E2 24399.18} C_VEL
LIN {X 0,Y 607.916,Z 780.356,A -85,B 0,C 180,E1 24397.086,E2 24397.086} C_VEL
LIN {X 0,Y 607.916,Z 784.639,A -85,B 0,C 180,E1 24395.001,E2 24395.001} C_VEL
LIN {X 0,Y 607.917,Z 787.517,A -85,B 0,C 180,E1 24392.923,E2 24392.923} C_VEL
LIN {X 0,Y 607.902,Z 788.828,A -85,B 0,C 180,E1 24390.754,E2 24390.754} C_VEL
LIN {X 0,Y 607.913,Z 788.694,A -85,B 0,C 180,E1 24388.681,E2 24388.681} C_VEL
LIN {X 0,Y 607.904,Z 786.953,A -85,B 0,C 180,E1 24386.606,E2 24386.606} C_VEL
LIN {X 0,Y 607.897,Z 783.842,A -85,B 0,C 180,E1 24384.526,E2 24384.526} C_VEL
LIN {X 0,Y 607.911,Z 779.08,A -85,B 0,C 180,E1 24382.439,E2 24382.439} C_VEL
LIN {X 0,Y 607.896,Z 773.428,A -85,B 0,C 180,E1 24380.533,E2 24380.533} C_VEL
LIN {X 0,Y 607.906,Z 765.149,A -85,B 0,C 180,E1 24378.329,E2 24378.329} C_VEL
LIN {X 0,Y 607.903,Z 756.364,A -85,B 0,C 180,E1 24376.397,E2 24376.397} C_VEL
LIN {X 0,Y 607.897,Z 745.296,A -85,B 0,C 180,E1 24374.351,E2 24374.351} C_VEL
LIN {X 0,Y 607.906,Z 733.591,A -85,B 0,C 180,E1 24372.483,E2 24372.483} C_VEL
LIN {X 0,Y 607.916,Z 719.886,A -85,B 0,C 180,E1 24370.596,E2 24370.596} C_VEL
LIN {X 0,Y 607.918,Z 704.989,A -85,B 0,C 180,E1 24368.787,E2 24368.787} C_VEL
LIN {X 0,Y 607.908,Z 688.59,A -85,B 0,C 180,E1 24367.058,E2 24367.058} C_VEL
LIN {X 0,Y 607.914,Z 670.217,A -85,B 0,C 180,E1 24365.359,E2 24365.359} C_VEL
LIN {X 0,Y 607.916,Z 651.609,A -85,B 0,C 180,E1 24363.847,E2 24363.847} C_VEL
LIN {X 0,Y 607.915,Z 631.971,A -85,B 0,C 180,E1 24362.474,E2 24362.474} C_VEL
LIN {X 0,Y 607.916,Z 610.806,A -85,B 0,C 180,E1 24361.191,E2 24361.191} C_VEL
LIN {X 0,Y 607.919,Z 591.964,A -85,B 0,C 180,E1 24360.219,E2 24360.219} C_VEL
LIN {X 0,Y 607.913,Z 570.035,A -85,B 0,C 180,E1 24359.262,E2 24359.262} C_VEL
LIN {X 0,Y 607.919,Z 550.614,A -85,B 0,C 180,E1 24358.576,E2 24358.576} C_VEL
LIN {X 0,Y 607.918,Z 530.246,A -85,B 0,C 180,E1 24357.995,E2 24357.995} C_VEL
LIN {X 0,Y 607.914,Z 509.002,A -85,B 0,C 180,E1 24357.557,E2 24357.557} C_VEL
LIN {X 0,Y 607.917,Z 278.293,A -85,B 0,C 180,E1 24354.309,E2 24354.309} C_VEL
LIN {X 0,Y 607.918,Z 160.96,A -85,B 0,C 180,E1 24352.599,E2 24352.599} C_VEL
LIN {X 0,Y 607.905,Z 126.831,A -85,B 0,C 180,E1 24350.507,E2 24350.507} C_VEL
LIN {X 0,Y 607.9,Z 126.342,A -85,B 0,C 180,E1 24350.332,E2 24350.332} C_VEL
LIN {X 0,Y 607.896,Z 126.321,A -85,B 0,C 180,E1 24347.187,E2 24347.187} C_VEL
LIN {X 0,Y 607.9,Z 126.319,A -85,B 0,C 180,E1 24344.049,E2 24344.049} C_VEL
LIN {X 0,Y 607.913,Z 126.327,A -85,B 0,C 180,E1 24340.765,E2 24340.765} C_VEL
LIN {X 0,Y 607.906,Z 126.319,A -85,B 0,C 180,E1 24337.485,E2 24337.485} C_VEL
LIN {X 0,Y 607.891,Z 126.323,A -85,B 0,C 180,E1 24334.344,E2 24334.344} C_VEL
LIN {X 0,Y 607.904,Z 126.322,A -85,B 0,C 180,E1 24331.205,E2 24331.205} C_VEL
LIN {X 0,Y 607.89,Z 126.319,A -85,B 0,C 180,E1 24328.061,E2 24328.061} C_VEL
LIN {X 0,Y 607.908,Z 126.327,A -85,B 0,C 180,E1 24324.786,E2 24324.786} C_VEL
LIN {X 0,Y 607.914,Z 126.317,A -85,B 0,C 180,E1 24321.517,E2 24321.517} C_VEL
LIN {X 0,Y 607.882,Z 126.323,A -85,B 0,C 180,E1 24318.371,E2 24318.371} C_VEL
LIN {X 0,Y 607.91,Z 126.321,A -85,B 0,C 180,E1 24315.257,E2 24315.257} C_VEL
LIN {X 0,Y 607.876,Z 126.322,A -85,B 0,C 180,E1 24312.154,E2 24312.154} C_VEL
LIN {X 0,Y 607.918,Z 126.327,A -85,B 0,C 180,E1 24308.989,E2 24308.989} C_VEL
LIN {X 0,Y 607.887,Z 126.32,A -85,B 0,C 180,E1 24305.853,E2 24305.853} C_VEL
LIN {X 0,Y 607.877,Z 126.325,A -85,B 0,C 180,E1 24302.545,E2 24302.545} C_VEL
LIN {X 0,Y 607.917,Z 126.32,A -85,B 0,C 180,E1 24299.434,E2 24299.434} C_VEL
LIN {X 0,Y 607.886,Z 126.326,A -85,B 0,C 180,E1 24296.73,E2 24296.73} C_VEL
LIN {X 0,Y 606.861,Z 126.451,A -85,B 0,C 180,E1 24296.004,E2 24296.004} C_VEL
LIN {X 0,Y 600.488,Z 127.244,A -85,B 0,C 180,E1 24293.968,E2 24293.968} C_VEL
LIN {X 0,Y 599.974,Z 127.31,A -85,B 0,C 180,E1 24293.438,E2 24293.438} C_VEL
LIN {X 0,Y 599.921,Z 127.313,A -85,B 0,C 180,E1 24290.309,E2 24290.309} C_VEL
LIN {X 0,Y 599.978,Z 127.315,A -85,B 0,C 180,E1 24287.128,E2 24287.128} C_VEL
LIN {X 0,Y 599.92,Z 127.313,A -85,B 0,C 180,E1 24284.038,E2 24284.038} C_VEL
LIN {X 0,Y 599.944,Z 127.313,A -85,B 0,C 180,E1 24280.833,E2 24280.833} C_VEL
LIN {X 0,Y 599.923,Z 127.313,A -85,B 0,C 180,E1 24277.873,E2 24277.873} C_VEL
LIN {X 0,Y 599.919,Z 127.313,A -85,B 0,C 180,E1 24274.596,E2 24274.596} C_VEL
LIN {X 0,Y 599.94,Z 127.314,A -85,B 0,C 180,E1 24271.635,E2 24271.635} C_VEL
LIN {X 0,Y 599.905,Z 127.314,A -85,B 0,C 180,E1 24268.443,E2 24268.443} C_VEL
LIN {X 0,Y 599.953,Z 127.315,A -85,B 0,C 180,E1 24265.484,E2 24265.484} C_VEL
LIN {X 0,Y 599.898,Z 127.316,A -85,B 0,C 180,E1 24262.409,E2 24262.409} C_VEL
LIN {X 0,Y 599.95,Z 127.314,A -85,B 0,C 180,E1 24259.458,E2 24259.458} C_VEL
LIN {X 0,Y 599.89,Z 127.315,A -85,B 0,C 180,E1 24256.331,E2 24256.331} C_VEL
LIN {X 0,Y 599.962,Z 127.316,A -85,B 0,C 180,E1 24253.361,E2 24253.361} C_VEL
LIN {X 0,Y 599.893,Z 127.318,A -85,B 0,C 180,E1 24250.238,E2 24250.238} C_VEL
LIN {X 0,Y 599.921,Z 127.476,A -85,B 0,C 180,E1 24248.071,E2 24248.071} C_VEL
LIN {X 0,Y 601.143,Z 130.863,A -85,B 0,C 180,E1 24247.697,E2 24247.697} C_VEL
LIN {X 0,Y 600.965,Z 175.011,A -85,B 0,C 180,E1 24244.86,E2 24244.86} C_VEL
LIN {X 0,Y 600.963,Z 209.265,A -85,B 0,C 180,E1 24242.741,E2 24242.741} C_VEL
LIN {X 0,Y 600.974,Z 363.618,A -85,B 0,C 180,E1 24240.613,E2 24240.613} C_VEL
LIN {X 0,Y 600.845,Z 514.373,A -85,B 0,C 180,E1 24238.561,E2 24238.561} C_VEL
LIN {X 0,Y 600.787,Z 535.322,A -85,B 0,C 180,E1 24238.104,E2 24238.104} C_VEL
LIN {X 0,Y 600.719,Z 556.245,A -85,B 0,C 180,E1 24237.483,E2 24237.483} C_VEL
LIN {X 0,Y 600.643,Z 576.292,A -85,B 0,C 180,E1 24236.708,E2 24236.708} C_VEL
LIN {X 0,Y 600.539,Z 597.408,A -85,B 0,C 180,E1 24235.703,E2 24235.703} C_VEL
LIN {X 0,Y 600.444,Z 616.734,A -85,B 0,C 180,E1 24234.6,E2 24234.6} C_VEL
LIN {X 0,Y 600.352,Z 635.896,A -85,B 0,C 180,E1 24233.299,E2 24233.299} C_VEL
LIN {X 0,Y 600.247,Z 653.526,A -85,B 0,C 180,E1 24231.902,E2 24231.902} C_VEL
LIN {X 0,Y 600.161,Z 670.214,A -85,B 0,C 180,E1 24230.376,E2 24230.376} C_VEL
LIN {X 0,Y 600.1,Z 685.588,A -85,B 0,C 180,E1 24228.757,E2 24228.757} C_VEL
LIN {X 0,Y 600.042,Z 700.266,A -85,B 0,C 180,E1 24226.954,E2 24226.954} C_VEL
LIN {X 0,Y 599.995,Z 712.754,A -85,B 0,C 180,E1 24225.166,E2 24225.166} C_VEL
LIN {X 0,Y 599.955,Z 724.092,A -85,B 0,C 180,E1 24223.277,E2 24223.277} C_VEL
LIN {X 0,Y 599.927,Z 733.349,A -85,B 0,C 180,E1 24221.439,E2 24221.439} C_VEL
LIN {X 0,Y 599.911,Z 741.8,A -85,B 0,C 180,E1 24219.4,E2 24219.4} C_VEL
LIN {X 0,Y 599.905,Z 748.51,A -85,B 0,C 180,E1 24217.373,E2 24217.373} C_VEL
LIN {X 0,Y 599.908,Z 753.213,A -85,B 0,C 180,E1 24215.451,E2 24215.451} C_VEL
LIN {X 0,Y 599.918,Z 756.819,A -85,B 0,C 180,E1 24213.312,E2 24213.312} C_VEL
LIN {X 0,Y 599.907,Z 758.683,A -85,B 0,C 180,E1 24211.241,E2 24211.241} C_VEL
LIN {X 0,Y 599.903,Z 758.839,A -85,B 0,C 180,E1 24209.236,E2 24209.236} C_VEL
LIN {X 0,Y 599.908,Z 757.448,A -85,B 0,C 180,E1 24207.134,E2 24207.134} C_VEL
LIN {X 0,Y 599.909,Z 754.561,A -85,B 0,C 180,E1 24205.124,E2 24205.124} C_VEL
LIN {X 0,Y 599.914,Z 750.017,A -85,B 0,C 180,E1 24203.108,E2 24203.108} C_VEL
LIN {X 0,Y 599.923,Z 743.904,A -85,B 0,C 180,E1 24201.084,E2 24201.084} C_VEL
LIN {X 0,Y 599.924,Z 736.346,A -85,B 0,C 180,E1 24199.145,E2 24199.145} C_VEL
LIN {X 0,Y 599.948,Z 726.548,A -85,B 0,C 180,E1 24197.096,E2 24197.096} C_VEL
LIN {X 0,Y 599.977,Z 715.901,A -85,B 0,C 180,E1 24195.228,E2 24195.228} C_VEL
LIN {X 0,Y 600.014,Z 703.335,A -85,B 0,C 180,E1 24193.371,E2 24193.371} C_VEL
LIN {X 0,Y 600.081,Z 689.75,A -85,B 0,C 180,E1 24191.645,E2 24191.645} C_VEL
LIN {X 0,Y 600.152,Z 674.149,A -85,B 0,C 180,E1 24189.929,E2 24189.929} C_VEL
LIN {X 0,Y 600.243,Z 657.619,A -85,B 0,C 180,E1 24188.356,E2 24188.356} C_VEL
LIN {X 0,Y 600.312,Z 639.883,A -85,B 0,C 180,E1 24186.907,E2 24186.907} C_VEL
LIN {X 0,Y 600.422,Z 621.333,A -85,B 0,C 180,E1 24185.608,E2 24185.608} C_VEL
LIN {X 0,Y 600.528,Z 602.083,A -85,B 0,C 180,E1 24184.455,E2 24184.455} C_VEL
LIN {X 0,Y 600.601,Z 583.141,A -85,B 0,C 180,E1 24183.503,E2 24183.503} C_VEL
LIN {X 0,Y 600.7,Z 562.446,A -85,B 0,C 180,E1 24182.653,E2 24182.653} C_VEL
LIN {X 0,Y 600.788,Z 541.76,A -85,B 0,C 180,E1 24181.974,E2 24181.974} C_VEL
LIN {X 0,Y 600.819,Z 521.177,A -85,B 0,C 180,E1 24181.481,E2 24181.481} C_VEL
LIN {X 0,Y 600.886,Z 494.659,A -85,B 0,C 180,E1 24181.06,E2 24181.06} C_VEL
LIN {X 0,Y 601.065,Z 269.261,A -85,B 0,C 180,E1 24178.01,E2 24178.01} C_VEL
LIN {X 0,Y 600.981,Z 209.339,A -85,B 0,C 180,E1 24177.17,E2 24177.17} C_VEL
LIN {X 0,Y 601.034,Z 163.686,A -85,B 0,C 180,E1 24174.334,E2 24174.334} C_VEL
LIN {X 0,Y 601.107,Z 130.624,A -85,B 0,C 180,E1 24172.195,E2 24172.195} C_VEL
LIN {X 0,Y 599.932,Z 127.505,A -85,B 0,C 180,E1 24171.851,E2 24171.851} C_VEL
LIN {X 0,Y 599.936,Z 127.316,A -85,B 0,C 180,E1 24169.084,E2 24169.084} C_VEL
LIN {X 0,Y 599.902,Z 127.317,A -85,B 0,C 180,E1 24165.919,E2 24165.919} C_VEL
LIN {X 0,Y 599.944,Z 127.314,A -85,B 0,C 180,E1 24162.972,E2 24162.972} C_VEL
LIN {X 0,Y 599.893,Z 127.315,A -85,B 0,C 180,E1 24159.918,E2 24159.918} C_VEL
LIN {X 0,Y 599.932,Z 127.317,A -85,B 0,C 180,E1 24157.033,E2 24157.033} C_VEL
LIN {X 0,Y 599.896,Z 127.316,A -85,B 0,C 180,E1 24153.901,E2 24153.901} C_VEL
LIN {X 0,Y 599.943,Z 127.315,A -85,B 0,C 180,E1 24150.996,E2 24150.996} C_VEL
LIN {X 0,Y 599.903,Z 127.315,A -85,B 0,C 180,E1 24147.927,E2 24147.927} C_VEL
LIN {X 0,Y 599.957,Z 127.314,A -85,B 0,C 180,E1 24144.938,E2 24144.938} C_VEL
LIN {X 0,Y 599.906,Z 127.315,A -85,B 0,C 180,E1 24141.819,E2 24141.819} C_VEL
LIN {X 0,Y 599.975,Z 127.313,A -85,B 0,C 180,E1 24138.762,E2 24138.762} C_VEL
LIN {X 0,Y 599.911,Z 127.314,A -85,B 0,C 180,E1 24135.665,E2 24135.665} C_VEL
LIN {X 0,Y 599.971,Z 127.311,A -85,B 0,C 180,E1 24132.512,E2 24132.512} C_VEL
LIN {X 0,Y 599.922,Z 127.314,A -85,B 0,C 180,E1 24129.497,E2 24129.497} C_VEL
LIN {X 0,Y 599.952,Z 127.311,A -85,B 0,C 180,E1 24126.315,E2 24126.315} C_VEL
LIN {X 0,Y 599.944,Z 127.314,A -85,B 0,C 180,E1 24123.248,E2 24123.248} C_VEL
LIN {X 0,Y 599.931,Z 127.311,A -85,B 0,C 180,E1 24120,E2 24120} C_VEL
LIN {X 0,Y 599.975,Z 127.316,A -85,B 0,C 180,E1 24116.943,E2 24116.943} C_VEL
LIN {X 0,Y 599.931,Z 127.312,A -85,B 0,C 180,E1 24113.781,E2 24113.781} C_VEL
LIN {X 0,Y 599.974,Z 127.311,A -85,B 0,C 180,E1 24110.697,E2 24110.697} C_VEL
LIN {X 0,Y 599.939,Z 127.313,A -85,B 0,C 180,E1 24107.581,E2 24107.581} C_VEL
LIN {X 0,Y 599.972,Z 127.305,A -85,B 0,C 180,E1 24104.411,E2 24104.411} C_VEL
LIN {X 0,Y 599.973,Z 127.316,A -85,B 0,C 180,E1 24101.137,E2 24101.137} C_VEL
LIN {X 0,Y 599.946,Z 127.307,A -85,B 0,C 180,E1 24097.91,E2 24097.91} C_VEL
LIN {X 0,Y 599.968,Z 127.311,A -85,B 0,C 180,E1 24094.746,E2 24094.746} C_VEL
LIN {X 0,Y 599.951,Z 127.311,A -85,B 0,C 180,E1 24091.534,E2 24091.534} C_VEL
LIN {X 0,Y 599.977,Z 127.304,A -85,B 0,C 180,E1 24088.336,E2 24088.336} C_VEL
LIN {X 0,Y 599.971,Z 127.314,A -85,B 0,C 180,E1 24085.021,E2 24085.021} C_VEL
LIN {X 0,Y 599.954,Z 127.31,A -85,B 0,C 180,E1 24081.809,E2 24081.809} C_VEL
LIN {X 0,Y 599.961,Z 127.311,A -85,B 0,C 180,E1 24078.704,E2 24078.704} C_VEL
LIN {X 0,Y 599.961,Z 127.313,A -85,B 0,C 180,E1 24075.501,E2 24075.501} C_VEL
LIN {X 0,Y 599.974,Z 127.302,A -85,B 0,C 180,E1 24072.189,E2 24072.189} C_VEL
LIN {X 0,Y 600.002,Z 127.524,A -85,B 0,C 180,E1 24070.103,E2 24070.103} C_VEL
LIN {X 0,Y 601.077,Z 130.49,A -85,B 0,C 180,E1 24069.78,E2 24069.78} C_VEL
LIN {X 0,Y 601.328,Z 132.787,A -85,B 0,C 180,E1 24069.617,E2 24069.617} C_VEL
LIN {X 0,Y 601.358,Z 162.115,A -85,B 0,C 180,E1 24067.843,E2 24067.843} C_VEL
LIN {X 0,Y 601.422,Z 269.344,A -85,B 0,C 180,E1 24066.266,E2 24066.266} C_VEL
LIN {X 0,Y 601.188,Z 479.514,A -85,B 0,C 180,E1 24063.288,E2 24063.288} C_VEL
LIN {X 0,Y 601.128,Z 514.865,A -85,B 0,C 180,E1 24062.753,E2 24062.753} C_VEL
LIN {X 0,Y 601.06,Z 536.475,A -85,B 0,C 180,E1 24062.246,E2 24062.246} C_VEL
LIN {X 0,Y 600.992,Z 557.872,A -85,B 0,C 180,E1 24061.592,E2 24061.592} C_VEL
LIN {X 0,Y 600.871,Z 578.693,A -85,B 0,C 180,E1 24060.775,E2 24060.775} C_VEL
LIN {X 0,Y 600.785,Z 598.676,A -85,B 0,C 180,E1 24059.841,E2 24059.841} C_VEL
LIN {X 0,Y 600.644,Z 619.4,A -85,B 0,C 180,E1 24058.686,E2 24058.686} C_VEL
LIN {X 0,Y 600.55,Z 639.116,A -85,B 0,C 180,E1 24057.414,E2 24057.414} C_VEL
LIN {X 0,Y 600.411,Z 658.265,A -85,B 0,C 180,E1 24055.974,E2 24055.974} C_VEL
LIN {X 0,Y 600.297,Z 677.253,A -85,B 0,C 180,E1 24054.345,E2 24054.345} C_VEL
LIN {X 0,Y 600.209,Z 693.66,A -85,B 0,C 180,E1 24052.735,E2 24052.735} C_VEL
LIN {X 0,Y 600.127,Z 709.29,A -85,B 0,C 180,E1 24050.989,E2 24050.989} C_VEL
LIN {X 0,Y 600.075,Z 723.964,A -85,B 0,C 180,E1 24049.136,E2 24049.136} C_VEL
LIN {X 0,Y 600.021,Z 736.808,A -85,B 0,C 180,E1 24047.254,E2 24047.254} C_VEL
LIN {X 0,Y 599.97,Z 748.933,A -85,B 0,C 180,E1 24045.224,E2 24045.224} C_VEL
LIN {X 0,Y 599.947,Z 758.784,A -85,B 0,C 180,E1 24043.275,E2 24043.275} C_VEL
LIN {X 0,Y 599.934,Z 767.912,A -85,B 0,C 180,E1 24041.147,E2 24041.147} C_VEL
LIN {X 0,Y 599.922,Z 774.953,A -85,B 0,C 180,E1 24039.11,E2 24039.11} C_VEL
LIN {X 0,Y 599.916,Z 781.014,A -85,B 0,C 180,E1 24036.892,E2 24036.892} C_VEL
LIN {X 0,Y 599.907,Z 784.957,A -85,B 0,C 180,E1 24034.876,E2 24034.876} C_VEL
LIN {X 0,Y 599.917,Z 787.786,A -85,B 0,C 180,E1 24032.675,E2 24032.675} C_VEL
LIN {X 0,Y 599.897,Z 788.872,A -85,B 0,C 180,E1 24030.573,E2 24030.573} C_VEL
LIN {X 0,Y 599.898,Z 788.524,A -85,B 0,C 180,E1 24028.376,E2 24028.376} C_VEL
LIN {X 0,Y 599.907,Z 786.728,A -85,B 0,C 180,E1 24026.369,E2 24026.369} C_VEL
LIN {X 0,Y 599.907,Z 783.287,A -85,B 0,C 180,E1 24024.165,E2 24024.165} C_VEL
LIN {X 0,Y 599.918,Z 778.57,A -85,B 0,C 180,E1 24022.145,E2 24022.145} C_VEL
LIN {X 0,Y 599.925,Z 772.184,A -85,B 0,C 180,E1 24020.019,E2 24020.019} C_VEL
LIN {X 0,Y 599.936,Z 764.332,A -85,B 0,C 180,E1 24017.976,E2 24017.976} C_VEL
LIN {X 0,Y 599.965,Z 754.913,A -85,B 0,C 180,E1 24015.91,E2 24015.91} C_VEL
LIN {X 0,Y 599.987,Z 744.136,A -85,B 0,C 180,E1 24013.941,E2 24013.941} C_VEL
LIN {X 0,Y 600.04,Z 731.584,A -85,B 0,C 180,E1 24011.945,E2 24011.945} C_VEL
LIN {X 0,Y 600.077,Z 718.331,A -85,B 0,C 180,E1 24010.129,E2 24010.129} C_VEL
LIN {X 0,Y 600.161,Z 702.201,A -85,B 0,C 180,E1 24008.192,E2 24008.192} C_VEL
LIN {X 0,Y 600.262,Z 685.538,A -85,B 0,C 180,E1 24006.437,E2 24006.437} C_VEL
LIN {X 0,Y 600.354,Z 667.802,A -85,B 0,C 180,E1 24004.817,E2 24004.817} C_VEL
LIN {X 0,Y 600.48,Z 647.389,A -85,B 0,C 180,E1 24003.188,E2 24003.188} C_VEL
LIN {X 0,Y 600.598,Z 627.95,A -85,B 0,C 180,E1 24001.839,E2 24001.839} C_VEL
LIN {X 0,Y 600.719,Z 607.829,A -85,B 0,C 180,E1 24000.649,E2 24000.649} C_VEL
LIN {X 0,Y 600.845,Z 586.74,A -85,B 0,C 180,E1 23999.575,E2 23999.575} C_VEL
LIN {X 0,Y 600.942,Z 565.687,A -85,B 0,C 180,E1 23998.7,E2 23998.7} C_VEL
LIN {X 0,Y 601.031,Z 544.184,A -85,B 0,C 180,E1 23997.965,E2 23997.965} C_VEL
LIN {X 0,Y 601.115,Z 522.32,A -85,B 0,C 180,E1 23997.408,E2 23997.408} C_VEL
LIN {X 0,Y 601.159,Z 502.49,A -85,B 0,C 180,E1 23997.039,E2 23997.039} C_VEL
LIN {X 0,Y 601.398,Z 285.101,A -85,B 0,C 180,E1 23993.96,E2 23993.96} C_VEL
LIN {X 0,Y 601.38,Z 162.247,A -85,B 0,C 180,E1 23992.161,E2 23992.161} C_VEL
LIN {X 0,Y 601.249,Z 152.615,A -85,B 0,C 180,E1 23991.603,E2 23991.603} C_VEL
LIN {X 0,Y 601.33,Z 130.898,A -85,B 0,C 180,E1 23990.266,E2 23990.266} C_VEL
LIN {X 0,Y 600.016,Z 127.622,A -85,B 0,C 180,E1 23989.915,E2 23989.915} C_VEL
LIN {X 0,Y 599.957,Z 127.285,A -85,B 0,C 180,E1 23989.085,E2 23989.085} C_VEL
LIN {X 0,Y 599.974,Z 127.308,A -85,B 0,C 180,E1 23985.847,E2 23985.847} C_VEL
LIN {X 0,Y 599.965,Z 127.314,A -85,B 0,C 180,E1 23982.559,E2 23982.559} C_VEL
LIN {X 0,Y 599.962,Z 127.31,A -85,B 0,C 180,E1 23979.353,E2 23979.353} C_VEL
LIN {X 0,Y 599.953,Z 127.31,A -85,B 0,C 180,E1 23976.236,E2 23976.236} C_VEL
LIN {X 0,Y 599.969,Z 127.314,A -85,B 0,C 180,E1 23973.021,E2 23973.021} C_VEL
LIN {X 0,Y 599.972,Z 127.307,A -85,B 0,C 180,E1 23969.747,E2 23969.747} C_VEL
LIN {X 0,Y 599.953,Z 127.313,A -85,B 0,C 180,E1 23966.502,E2 23966.502} C_VEL
LIN {X 0,Y 599.969,Z 127.31,A -85,B 0,C 180,E1 23963.332,E2 23963.332} C_VEL
LIN {X 0,Y 599.943,Z 127.31,A -85,B 0,C 180,E1 23960.181,E2 23960.181} C_VEL
LIN {X 0,Y 599.974,Z 127.316,A -85,B 0,C 180,E1 23956.953,E2 23956.953} C_VEL
LIN {X 0,Y 599.968,Z 127.306,A -85,B 0,C 180,E1 23953.689,E2 23953.689} C_VEL
LIN {X 0,Y 599.941,Z 127.313,A -85,B 0,C 180,E1 23950.466,E2 23950.466} C_VEL
LIN {X 0,Y 599.975,Z 127.31,A -85,B 0,C 180,E1 23947.372,E2 23947.372} C_VEL
LIN {X 0,Y 599.932,Z 127.311,A -85,B 0,C 180,E1 23944.205,E2 23944.205} C_VEL
LIN {X 0,Y 599.974,Z 127.316,A -85,B 0,C 180,E1 23941.05,E2 23941.05} C_VEL
LIN {X 0,Y 599.939,Z 127.311,A -85,B 0,C 180,E1 23937.899,E2 23937.899} C_VEL
LIN {X 0,Y 599.939,Z 127.315,A -85,B 0,C 180,E1 23934.645,E2 23934.645} C_VEL
LIN {X 0,Y 599.974,Z 127.31,A -85,B 0,C 180,E1 23933.438,E2 23933.438} C_VEL
LIN {X 0,Y 598.988,Z 127.439,A -85,B 0,C 180,E1 23932.702,E2 23932.702} C_VEL
LIN {X 0,Y 592.51,Z 128.241,A -85,B 0,C 180,E1 23930.638,E2 23930.638} C_VEL
LIN {X 0,Y 591.985,Z 128.301,A -85,B 0,C 180,E1 23930.101,E2 23930.101} C_VEL
LIN {X 0,Y 592.02,Z 128.304,A -85,B 0,C 180,E1 23926.92,E2 23926.92} C_VEL
LIN {X 0,Y 591.987,Z 128.302,A -85,B 0,C 180,E1 23923.919,E2 23923.919} C_VEL
LIN {X 0,Y 591.983,Z 128.3,A -85,B 0,C 180,E1 23920.565,E2 23920.565} C_VEL
LIN {X 0,Y 592.023,Z 128.301,A -85,B 0,C 180,E1 23917.487,E2 23917.487} C_VEL
LIN {X 0,Y 591.971,Z 128.3,A -85,B 0,C 180,E1 23914.38,E2 23914.38} C_VEL
LIN {X 0,Y 592.04,Z 128.305,A -85,B 0,C 180,E1 23911.221,E2 23911.221} C_VEL
LIN {X 0,Y 591.964,Z 128.302,A -85,B 0,C 180,E1 23908.165,E2 23908.165} C_VEL
LIN {X 0,Y 592.021,Z 128.301,A -85,B 0,C 180,E1 23905.073,E2 23905.073} C_VEL
LIN {X 0,Y 591.96,Z 128.306,A -85,B 0,C 180,E1 23902.061,E2 23902.061} C_VEL
LIN {X 0,Y 591.989,Z 128.307,A -85,B 0,C 180,E1 23898.874,E2 23898.874} C_VEL
LIN {X 0,Y 591.956,Z 128.303,A -85,B 0,C 180,E1 23896.015,E2 23896.015} C_VEL
LIN {X 0,Y 591.975,Z 128.3,A -85,B 0,C 180,E1 23892.763,E2 23892.763} C_VEL
LIN {X 0,Y 591.964,Z 128.308,A -85,B 0,C 180,E1 23889.928,E2 23889.928} C_VEL
LIN {X 0,Y 592.007,Z 128.583,A -85,B 0,C 180,E1 23888.578,E2 23888.578} C_VEL
LIN {X 0,Y 594.404,Z 134.549,A -85,B 0,C 180,E1 23887.955,E2 23887.955} C_VEL
LIN {X 0,Y 594.031,Z 179.695,A -85,B 0,C 180,E1 23885.026,E2 23885.026} C_VEL
LIN {X 0,Y 593.964,Z 209.402,A -85,B 0,C 180,E1 23883.174,E2 23883.174} C_VEL
LIN {X 0,Y 594.405,Z 213.831,A -85,B 0,C 180,E1 23883.081,E2 23883.081} C_VEL
LIN {X 0,Y 593.969,Z 444.586,A -85,B 0,C 180,E1 23879.901,E2 23879.901} C_VEL
LIN {X 0,Y 593.81,Z 515.487,A -85,B 0,C 180,E1 23878.914,E2 23878.914} C_VEL
LIN {X 0,Y 593.689,Z 536.422,A -85,B 0,C 180,E1 23878.442,E2 23878.442} C_VEL
LIN {X 0,Y 593.531,Z 557.803,A -85,B 0,C 180,E1 23877.788,E2 23877.788} C_VEL
LIN {X 0,Y 593.388,Z 577.585,A -85,B 0,C 180,E1 23877.007,E2 23877.007} C_VEL
LIN {X 0,Y 593.182,Z 597.357,A -85,B 0,C 180,E1 23876.049,E2 23876.049} C_VEL
LIN {X 0,Y 593.003,Z 616.742,A -85,B 0,C 180,E1 23874.93,E2 23874.93} C_VEL
LIN {X 0,Y 592.804,Z 635.181,A -85,B 0,C 180,E1 23873.667,E2 23873.667} C_VEL
LIN {X 0,Y 592.599,Z 653.468,A -85,B 0,C 180,E1 23872.206,E2 23872.206} C_VEL
LIN {X 0,Y 592.419,Z 670.726,A -85,B 0,C 180,E1 23870.603,E2 23870.603} C_VEL
LIN {X 0,Y 592.298,Z 685.594,A -85,B 0,C 180,E1 23869.014,E2 23869.014} C_VEL
LIN {X 0,Y 592.174,Z 700.272,A -85,B 0,C 180,E1 23867.186,E2 23867.186} C_VEL
LIN {X 0,Y 592.072,Z 712.844,A -85,B 0,C 180,E1 23865.361,E2 23865.361} C_VEL
LIN {X 0,Y 592,Z 723.999,A -85,B 0,C 180,E1 23863.478,E2 23863.478} C_VEL
LIN {X 0,Y 591.954,Z 733.455,A -85,B 0,C 180,E1 23861.573,E2 23861.573} C_VEL
LIN {X 0,Y 591.922,Z 741.802,A -85,B 0,C 180,E1 23859.528,E2 23859.528} C_VEL
LIN {X 0,Y 591.912,Z 748.245,A -85,B 0,C 180,E1 23857.571,E2 23857.571} C_VEL
LIN {X 0,Y 591.912,Z 753.214,A -85,B 0,C 180,E1 23855.525,E2 23855.525} C_VEL
LIN {X 0,Y 591.917,Z 756.85,A -85,B 0,C 180,E1 23853.331,E2 23853.331} C_VEL
LIN {X 0,Y 591.906,Z 758.683,A -85,B 0,C 180,E1 23851.258,E2 23851.258} C_VEL
LIN {X 0,Y 591.904,Z 758.839,A -85,B 0,C 180,E1 23849.226,E2 23849.226} C_VEL
LIN {X 0,Y 591.91,Z 757.448,A -85,B 0,C 180,E1 23847.095,E2 23847.095} C_VEL
LIN {X 0,Y 591.913,Z 754.561,A -85,B 0,C 180,E1 23845.058,E2 23845.058} C_VEL
LIN {X 0,Y 591.918,Z 750.016,A -85,B 0,C 180,E1 23843.015,E2 23843.015} C_VEL
LIN {X 0,Y 591.939,Z 743.901,A -85,B 0,C 180,E1 23840.962,E2 23840.962} C_VEL
LIN {X 0,Y 591.953,Z 736.345,A -85,B 0,C 180,E1 23838.997,E2 23838.997} C_VEL
LIN {X 0,Y 591.997,Z 726.546,A -85,B 0,C 180,E1 23836.92,E2 23836.92} C_VEL
LIN {X 0,Y 592.061,Z 715.807,A -85,B 0,C 180,E1 23835.012,E2 23835.012} C_VEL
LIN {X 0,Y 592.13,Z 703.854,A -85,B 0,C 180,E1 23833.218,E2 23833.218} C_VEL
LIN {X 0,Y 592.256,Z 689.745,A -85,B 0,C 180,E1 23831.394,E2 23831.394} C_VEL
LIN {X 0,Y 592.404,Z 674.143,A -85,B 0,C 180,E1 23829.655,E2 23829.655} C_VEL
LIN {X 0,Y 592.58,Z 657.261,A -85,B 0,C 180,E1 23828.031,E2 23828.031} C_VEL
LIN {X 0,Y 592.762,Z 639.207,A -85,B 0,C 180,E1 23826.543,E2 23826.543} C_VEL
LIN {X 0,Y 592.94,Z 620.523,A -85,B 0,C 180,E1 23825.227,E2 23825.227} C_VEL
LIN {X 0,Y 593.168,Z 600.085,A -85,B 0,C 180,E1 23824.008,E2 23824.008} C_VEL
LIN {X 0,Y 593.355,Z 580.868,A -85,B 0,C 180,E1 23823.046,E2 23823.046} C_VEL
LIN {X 0,Y 593.52,Z 560.228,A -85,B 0,C 180,E1 23822.212,E2 23822.212} C_VEL
LIN {X 0,Y 593.686,Z 537.974,A -85,B 0,C 180,E1 23821.509,E2 23821.509} C_VEL
LIN {X 0,Y 593.78,Z 517.445,A -85,B 0,C 180,E1 23821.032,E2 23821.032} C_VEL
LIN {X 0,Y 593.899,Z 481.246,A -85,B 0,C 180,E1 23820.505,E2 23820.505} C_VEL
LIN {X 0,Y 594.302,Z 253.426,A -85,B 0,C 180,E1 23817.38,E2 23817.38} C_VEL
LIN {X 0,Y 594.217,Z 210.762,A -85,B 0,C 180,E1 23816.773,E2 23816.773} C_VEL
LIN {X 0,Y 593.855,Z 208.168,A -85,B 0,C 180,E1 23816.682,E2 23816.682} C_VEL
LIN {X 0,Y 594.242,Z 156.261,A -85,B 0,C 180,E1 23813.378,E2 23813.378} C_VEL
LIN {X 0,Y 594.327,Z 134.37,A -85,B 0,C 180,E1 23811.937,E2 23811.937} C_VEL
LIN {X 0,Y 592.011,Z 128.537,A -85,B 0,C 180,E1 23811.326,E2 23811.326} C_VEL
LIN {X 0,Y 592.029,Z 128.301,A -85,B 0,C 180,E1 23808.578,E2 23808.578} C_VEL
LIN {X 0,Y 591.959,Z 128.307,A -85,B 0,C 180,E1 23805.6,E2 23805.6} C_VEL
LIN {X 0,Y 592.011,Z 128.307,A -85,B 0,C 180,E1 23802.498,E2 23802.498} C_VEL
LIN {X 0,Y 591.953,Z 128.303,A -85,B 0,C 180,E1 23799.553,E2 23799.553} C_VEL
LIN {X 0,Y 592.004,Z 128.3,A -85,B 0,C 180,E1 23796.478,E2 23796.478} C_VEL
LIN {X 0,Y 591.962,Z 128.306,A -85,B 0,C 180,E1 23793.45,E2 23793.45} C_VEL
LIN {X 0,Y 591.976,Z 128.302,A -85,B 0,C 180,E1 23790.146,E2 23790.146} C_VEL
LIN {X 0,Y 591.982,Z 128.305,A -85,B 0,C 180,E1 23787.24,E2 23787.24} C_VEL
LIN {X 0,Y 591.971,Z 128.302,A -85,B 0,C 180,E1 23783.972,E2 23783.972} C_VEL
LIN {X 0,Y 592.017,Z 128.305,A -85,B 0,C 180,E1 23780.98,E2 23780.98} C_VEL
LIN {X 0,Y 591.971,Z 128.301,A -85,B 0,C 180,E1 23777.801,E2 23777.801} C_VEL
LIN {X 0,Y 592.041,Z 128.301,A -85,B 0,C 180,E1 23774.674,E2 23774.674} C_VEL
LIN {X 0,Y 591.978,Z 128.303,A -85,B 0,C 180,E1 23771.593,E2 23771.593} C_VEL
LIN {X 0,Y 592.026,Z 128.299,A -85,B 0,C 180,E1 23768.449,E2 23768.449} C_VEL
LIN {X 0,Y 591.997,Z 128.304,A -85,B 0,C 180,E1 23765.33,E2 23765.33} C_VEL
LIN {X 0,Y 591.994,Z 128.301,A -85,B 0,C 180,E1 23762.033,E2 23762.033} C_VEL
LIN {X 0,Y 592.034,Z 128.306,A -85,B 0,C 180,E1 23758.936,E2 23758.936} C_VEL
LIN {X 0,Y 591.991,Z 128.301,A -85,B 0,C 180,E1 23755.738,E2 23755.738} C_VEL
LIN {X 0,Y 592.039,Z 128.297,A -85,B 0,C 180,E1 23752.528,E2 23752.528} C_VEL
LIN {X 0,Y 592.013,Z 128.303,A -85,B 0,C 180,E1 23749.294,E2 23749.294} C_VEL
LIN {X 0,Y 592.006,Z 128.296,A -85,B 0,C 180,E1 23746.024,E2 23746.024} C_VEL
LIN {X 0,Y 592.033,Z 128.302,A -85,B 0,C 180,E1 23742.81,E2 23742.81} C_VEL
LIN {X 0,Y 592.004,Z 128.3,A -85,B 0,C 180,E1 23739.64,E2 23739.64} C_VEL
LIN {X 0,Y 592.038,Z 128.296,A -85,B 0,C 180,E1 23736.406,E2 23736.406} C_VEL
LIN {X 0,Y 592.034,Z 128.3,A -85,B 0,C 180,E1 23733.086,E2 23733.086} C_VEL
LIN {X 0,Y 592.012,Z 128.3,A -85,B 0,C 180,E1 23729.848,E2 23729.848} C_VEL
LIN {X 0,Y 592.026,Z 128.3,A -85,B 0,C 180,E1 23726.71,E2 23726.71} C_VEL
LIN {X 0,Y 592.02,Z 128.301,A -85,B 0,C 180,E1 23723.503,E2 23723.503} C_VEL
LIN {X 0,Y 592.036,Z 128.295,A -85,B 0,C 180,E1 23720.203,E2 23720.203} C_VEL
LIN {X 0,Y 592.025,Z 128.301,A -85,B 0,C 180,E1 23716.976,E2 23716.976} C_VEL
LIN {X 0,Y 592.021,Z 128.302,A -85,B 0,C 180,E1 23713.822,E2 23713.822} C_VEL
LIN {X 0,Y 592.025,Z 128.342,A -85,B 0,C 180,E1 23710.748,E2 23710.748} C_VEL
LIN {X 0,Y 592.256,Z 129.447,A -85,B 0,C 180,E1 23710.563,E2 23710.563} C_VEL
LIN {X 0,Y 594.766,Z 134.983,A -85,B 0,C 180,E1 23710.002,E2 23710.002} C_VEL
LIN {X 0,Y 594.694,Z 162.115,A -85,B 0,C 180,E1 23708.344,E2 23708.344} C_VEL
LIN {X 0,Y 595.215,Z 166.37,A -85,B 0,C 180,E1 23708.24,E2 23708.24} C_VEL
LIN {X 0,Y 594.731,Z 374.148,A -85,B 0,C 180,E1 23705.209,E2 23705.209} C_VEL
LIN {X 0,Y 594.413,Z 510.409,A -85,B 0,C 180,E1 23703.25,E2 23703.25} C_VEL
LIN {X 0,Y 594.251,Z 534.144,A -85,B 0,C 180,E1 23702.725,E2 23702.725} C_VEL
LIN {X 0,Y 594.115,Z 554.065,A -85,B 0,C 180,E1 23702.127,E2 23702.127} C_VEL
LIN {X 0,Y 593.861,Z 577.424,A -85,B 0,C 180,E1 23701.235,E2 23701.235} C_VEL
LIN {X 0,Y 593.682,Z 597.561,A -85,B 0,C 180,E1 23700.291,E2 23700.291} C_VEL
LIN {X 0,Y 593.398,Z 619.158,A -85,B 0,C 180,E1 23699.085,E2 23699.085} C_VEL
LIN {X 0,Y 593.2,Z 639.438,A -85,B 0,C 180,E1 23697.761,E2 23697.761} C_VEL
LIN {X 0,Y 592.93,Z 658.267,A -85,B 0,C 180,E1 23696.326,E2 23696.326} C_VEL
LIN {X 0,Y 592.703,Z 677.33,A -85,B 0,C 180,E1 23694.67,E2 23694.67} C_VEL
LIN {X 0,Y 592.524,Z 694.356,A -85,B 0,C 180,E1 23692.974,E2 23692.974} C_VEL
LIN {X 0,Y 592.352,Z 710.143,A -85,B 0,C 180,E1 23691.175,E2 23691.175} C_VEL
LIN {X 0,Y 592.236,Z 724.587,A -85,B 0,C 180,E1 23689.31,E2 23689.31} C_VEL
LIN {X 0,Y 592.126,Z 737.452,A -85,B 0,C 180,E1 23687.39,E2 23687.39} C_VEL
LIN {X 0,Y 592.029,Z 749.753,A -85,B 0,C 180,E1 23685.275,E2 23685.275} C_VEL
LIN {X 0,Y 591.982,Z 759.15,A -85,B 0,C 180,E1 23683.379,E2 23683.379} C_VEL
LIN {X 0,Y 591.95,Z 768.626,A -85,B 0,C 180,E1 23681.102,E2 23681.102} C_VEL
LIN {X 0,Y 591.93,Z 775.259,A -85,B 0,C 180,E1 23679.136,E2 23679.136} C_VEL
LIN {X 0,Y 591.917,Z 781.427,A -85,B 0,C 180,E1 23676.791,E2 23676.791} C_VEL
LIN {X 0,Y 591.905,Z 785.117,A -85,B 0,C 180,E1 23674.845,E2 23674.845} C_VEL
LIN {X 0,Y 591.917,Z 787.853,A -85,B 0,C 180,E1 23672.614,E2 23672.614} C_VEL
LIN {X 0,Y 591.897,Z 788.872,A -85,B 0,C 180,E1 23670.581,E2 23670.581} C_VEL
LIN {X 0,Y 591.898,Z 788.524,A -85,B 0,C 180,E1 23668.354,E2 23668.354} C_VEL
LIN {X 0,Y 591.909,Z 786.728,A -85,B 0,C 180,E1 23666.32,E2 23666.32} C_VEL
LIN {X 0,Y 591.912,Z 783.287,A -85,B 0,C 180,E1 23664.086,E2 23664.086} C_VEL
LIN {X 0,Y 591.921,Z 778.571,A -85,B 0,C 180,E1 23662.038,E2 23662.038} C_VEL
LIN {X 0,Y 591.942,Z 772.183,A -85,B 0,C 180,E1 23659.883,E2 23659.883} C_VEL
LIN {X 0,Y 591.963,Z 764.333,A -85,B 0,C 180,E1 23657.812,E2 23657.812} C_VEL
LIN {X 0,Y 592.012,Z 754.954,A -85,B 0,C 180,E1 23655.725,E2 23655.725} C_VEL
LIN {X 0,Y 592.073,Z 744.138,A -85,B 0,C 180,E1 23653.721,E2 23653.721} C_VEL
LIN {X 0,Y 592.177,Z 731.582,A -85,B 0,C 180,E1 23651.697,E2 23651.697} C_VEL
LIN {X 0,Y 592.27,Z 718.074,A -85,B 0,C 180,E1 23649.822,E2 23649.822} C_VEL
LIN {X 0,Y 592.437,Z 701.737,A -85,B 0,C 180,E1 23647.84,E2 23647.84} C_VEL
LIN {X 0,Y 592.632,Z 685.538,A -85,B 0,C 180,E1 23646.115,E2 23646.115} C_VEL
LIN {X 0,Y 592.816,Z 667.729,A -85,B 0,C 180,E1 23644.467,E2 23644.467} C_VEL
LIN {X 0,Y 593.065,Z 648.309,A -85,B 0,C 180,E1 23642.894,E2 23642.894} C_VEL
LIN {X 0,Y 593.282,Z 629.569,A -85,B 0,C 180,E1 23641.57,E2 23641.57} C_VEL
LIN {X 0,Y 593.54,Z 608.826,A -85,B 0,C 180,E1 23640.314,E2 23640.314} C_VEL
LIN {X 0,Y 593.758,Z 588.604,A -85,B 0,C 180,E1 23639.265,E2 23639.265} C_VEL
LIN {X 0,Y 593.988,Z 567.23,A -85,B 0,C 180,E1 23638.351,E2 23638.351} C_VEL
LIN {X 0,Y 594.145,Z 546.199,A -85,B 0,C 180,E1 23637.615,E2 23637.615} C_VEL
LIN {X 0,Y 594.339,Z 523.455,A -85,B 0,C 180,E1 23637.015,E2 23637.015} C_VEL
LIN {X 0,Y 594.431,Z 503.775,A -85,B 0,C 180,E1 23636.639,E2 23636.639} C_VEL
LIN {X 0,Y 594.922,Z 285.738,A -85,B 0,C 180,E1 23633.514,E2 23633.514} C_VEL
LIN {X 0,Y 595.06,Z 163.963,A -85,B 0,C 180,E1 23631.712,E2 23631.712} C_VEL
LIN {X 0,Y 594.56,Z 160.759,A -85,B 0,C 180,E1 23631.597,E2 23631.597} C_VEL
LIN {X 0,Y 594.723,Z 134.84,A -85,B 0,C 180,E1 23629.985,E2 23629.985} C_VEL
LIN {X 0,Y 592.078,Z 128.677,A -85,B 0,C 180,E1 23629.342,E2 23629.342} C_VEL
LIN {X 0,Y 592.027,Z 128.259,A -85,B 0,C 180,E1 23628.871,E2 23628.871} C_VEL
LIN {X 0,Y 592.03,Z 128.299,A -85,B 0,C 180,E1 23625.593,E2 23625.593} C_VEL
LIN {X 0,Y 592.019,Z 128.302,A -85,B 0,C 180,E1 23622.366,E2 23622.366} C_VEL
LIN {X 0,Y 592.022,Z 128.301,A -85,B 0,C 180,E1 23619.171,E2 23619.171} C_VEL
LIN {X 0,Y 592.02,Z 128.297,A -85,B 0,C 180,E1 23615.996,E2 23615.996} C_VEL
LIN {X 0,Y 592.032,Z 128.3,A -85,B 0,C 180,E1 23612.713,E2 23612.713} C_VEL
LIN {X 0,Y 592.03,Z 128.298,A -85,B 0,C 180,E1 23609.436,E2 23609.436} C_VEL
LIN {X 0,Y 592.01,Z 128.299,A -85,B 0,C 180,E1 23606.26,E2 23606.26} C_VEL
LIN {X 0,Y 592.035,Z 128.304,A -85,B 0,C 180,E1 23603.016,E2 23603.016} C_VEL
LIN {X 0,Y 592.027,Z 128.295,A -85,B 0,C 180,E1 23599.741,E2 23599.741} C_VEL
LIN {X 0,Y 592.007,Z 128.298,A -85,B 0,C 180,E1 23596.483,E2 23596.483} C_VEL
LIN {X 0,Y 592.035,Z 128.296,A -85,B 0,C 180,E1 23593.378,E2 23593.378} C_VEL
LIN {X 0,Y 591.998,Z 128.299,A -85,B 0,C 180,E1 23590.215,E2 23590.215} C_VEL
LIN {X 0,Y 592.034,Z 128.304,A -85,B 0,C 180,E1 23586.984,E2 23586.984} C_VEL
LIN {X 0,Y 592.013,Z 128.298,A -85,B 0,C 180,E1 23583.777,E2 23583.777} C_VEL
LIN {X 0,Y 591.995,Z 128.302,A -85,B 0,C 180,E1 23580.484,E2 23580.484} C_VEL
LIN {X 0,Y 592.038,Z 128.301,A -85,B 0,C 180,E1 23577.289,E2 23577.289} C_VEL
LIN {X 0,Y 591.987,Z 128.301,A -85,B 0,C 180,E1 23574.146,E2 23574.146} C_VEL
LIN {X 0,Y 592.029,Z 128.305,A -85,B 0,C 180,E1 23570.963,E2 23570.963} C_VEL
LIN {X 0,Y 591.985,Z 128.301,A -85,B 0,C 180,E1 23570.101,E2 23570.101} C_VEL
LIN {X 0,Y 591.025,Z 128.427,A -85,B 0,C 180,E1 23569.355,E2 23569.355} C_VEL
LIN {X 0,Y 584.529,Z 129.24,A -85,B 0,C 180,E1 23567.209,E2 23567.209} C_VEL
LIN {X 0,Y 584.061,Z 129.292,A -85,B 0,C 180,E1 23566.719,E2 23566.719} C_VEL
LIN {X 0,Y 584.077,Z 129.29,A -85,B 0,C 180,E1 23563.593,E2 23563.593} C_VEL
LIN {X 0,Y 584.037,Z 129.287,A -85,B 0,C 180,E1 23560.394,E2 23560.394} C_VEL
LIN {X 0,Y 584.102,Z 129.292,A -85,B 0,C 180,E1 23557.24,E2 23557.24} C_VEL
LIN {X 0,Y 584.031,Z 129.287,A -85,B 0,C 180,E1 23554.115,E2 23554.115} C_VEL
LIN {X 0,Y 584.065,Z 129.292,A -85,B 0,C 180,E1 23550.91,E2 23550.91} C_VEL
LIN {X 0,Y 584.034,Z 129.29,A -85,B 0,C 180,E1 23547.931,E2 23547.931} C_VEL
LIN {X 0,Y 584.03,Z 129.287,A -85,B 0,C 180,E1 23544.576,E2 23544.576} C_VEL
LIN {X 0,Y 584.052,Z 129.295,A -85,B 0,C 180,E1 23541.632,E2 23541.632} C_VEL
LIN {X 0,Y 584.018,Z 129.296,A -85,B 0,C 180,E1 23538.429,E2 23538.429} C_VEL
LIN {X 0,Y 584.089,Z 129.288,A -85,B 0,C 180,E1 23535.286,E2 23535.286} C_VEL
LIN {X 0,Y 584.014,Z 129.288,A -85,B 0,C 180,E1 23532.152,E2 23532.152} C_VEL
LIN {X 0,Y 584.114,Z 129.465,A -85,B 0,C 180,E1 23529.156,E2 23529.156} C_VEL
LIN {X 0,Y 585.135,Z 132.432,A -85,B 0,C 180,E1 23528.813,E2 23528.813} C_VEL
LIN {X 0,Y 587.67,Z 138.145,A -85,B 0,C 180,E1 23528.226,E2 23528.226} C_VEL
LIN {X 0,Y 587.123,Z 182.745,A -85,B 0,C 180,E1 23525.301,E2 23525.301} C_VEL
LIN {X 0,Y 586.986,Z 209.453,A -85,B 0,C 180,E1 23523.62,E2 23523.62} C_VEL
LIN {X 0,Y 587.7,Z 214.703,A -85,B 0,C 180,E1 23523.497,E2 23523.497} C_VEL
LIN {X 0,Y 587.031,Z 445.975,A -85,B 0,C 180,E1 23520.273,E2 23520.273} C_VEL
LIN {X 0,Y 586.802,Z 515.636,A -85,B 0,C 180,E1 23519.291,E2 23519.291} C_VEL
LIN {X 0,Y 586.614,Z 536.71,A -85,B 0,C 180,E1 23518.81,E2 23518.81} C_VEL
LIN {X 0,Y 586.376,Z 558.41,A -85,B 0,C 180,E1 23518.135,E2 23518.135} C_VEL
LIN {X 0,Y 586.149,Z 578.875,A -85,B 0,C 180,E1 23517.313,E2 23517.313} C_VEL
LIN {X 0,Y 585.836,Z 598.434,A -85,B 0,C 180,E1 23516.342,E2 23516.342} C_VEL
LIN {X 0,Y 585.54,Z 618.371,A -85,B 0,C 180,E1 23515.162,E2 23515.162} C_VEL
LIN {X 0,Y 585.257,Z 637.373,A -85,B 0,C 180,E1 23513.83,E2 23513.83} C_VEL
LIN {X 0,Y 584.949,Z 655.08,A -85,B 0,C 180,E1 23512.371,E2 23512.371} C_VEL
LIN {X 0,Y 584.675,Z 672.251,A -85,B 0,C 180,E1 23510.731,E2 23510.731} C_VEL
LIN {X 0,Y 584.458,Z 688.153,A -85,B 0,C 180,E1 23508.968,E2 23508.968} C_VEL
LIN {X 0,Y 584.303,Z 701.81,A -85,B 0,C 180,E1 23507.219,E2 23507.219} C_VEL
LIN {X 0,Y 584.157,Z 714.688,A -85,B 0,C 180,E1 23505.283,E2 23505.283} C_VEL
LIN {X 0,Y 584.048,Z 726.08,A -85,B 0,C 180,E1 23503.261,E2 23503.261} C_VEL
LIN {X 0,Y 583.983,Z 735.568,A -85,B 0,C 180,E1 23501.255,E2 23501.255} C_VEL
LIN {X 0,Y 583.94,Z 743.224,A -85,B 0,C 180,E1 23499.262,E2 23499.262} C_VEL
LIN {X 0,Y 583.921,Z 749.529,A -85,B 0,C 180,E1 23497.181,E2 23497.181} C_VEL
LIN {X 0,Y 583.916,Z 754.242,A -85,B 0,C 180,E1 23495.108,E2 23495.108} C_VEL
LIN {X 0,Y 583.913,Z 757.232,A -85,B 0,C 180,E1 23493.043,E2 23493.043} C_VEL
LIN {X 0,Y 583.91,Z 758.796,A -85,B 0,C 180,E1 23490.883,E2 23490.883} C_VEL
LIN {X 0,Y 583.915,Z 758.749,A -85,B 0,C 180,E1 23488.823,E2 23488.823} C_VEL
LIN {X 0,Y 583.911,Z 757.111,A -85,B 0,C 180,E1 23486.761,E2 23486.761} C_VEL
LIN {X 0,Y 583.907,Z 754.021,A -85,B 0,C 180,E1 23484.695,E2 23484.695} C_VEL
LIN {X 0,Y 583.916,Z 749.506,A -85,B 0,C 180,E1 23482.721,E2 23482.721} C_VEL
LIN {X 0,Y 583.933,Z 742.836,A -85,B 0,C 180,E1 23480.539,E2 23480.539} C_VEL
LIN {X 0,Y 583.985,Z 735.12,A -85,B 0,C 180,E1 23478.545,E2 23478.545} C_VEL
LIN {X 0,Y 584.047,Z 725.505,A -85,B 0,C 180,E1 23476.537,E2 23476.537} C_VEL
LIN {X 0,Y 584.154,Z 713.916,A -85,B 0,C 180,E1 23474.505,E2 23474.505} C_VEL
LIN {X 0,Y 584.307,Z 701.719,A -85,B 0,C 180,E1 23472.678,E2 23472.678} C_VEL
LIN {X 0,Y 584.46,Z 688.039,A -85,B 0,C 180,E1 23470.929,E2 23470.929} C_VEL
LIN {X 0,Y 584.671,Z 672.617,A -85,B 0,C 180,E1 23469.216,E2 23469.216} C_VEL
LIN {X 0,Y 584.943,Z 655.711,A -85,B 0,C 180,E1 23467.594,E2 23467.594} C_VEL
LIN {X 0,Y 585.253,Z 637.854,A -85,B 0,C 180,E1 23466.116,E2 23466.116} C_VEL
LIN {X 0,Y 585.526,Z 618.912,A -85,B 0,C 180,E1 23464.784,E2 23464.784} C_VEL
LIN {X 0,Y 585.831,Z 599.083,A -85,B 0,C 180,E1 23463.603,E2 23463.603} C_VEL
LIN {X 0,Y 586.141,Z 579.686,A -85,B 0,C 180,E1 23462.632,E2 23462.632} C_VEL
LIN {X 0,Y 586.371,Z 558.743,A -85,B 0,C 180,E1 23461.787,E2 23461.787} C_VEL
LIN {X 0,Y 586.614,Z 536.781,A -85,B 0,C 180,E1 23461.102,E2 23461.102} C_VEL
LIN {X 0,Y 586.802,Z 515.683,A -85,B 0,C 180,E1 23460.62,E2 23460.62} C_VEL
LIN {X 0,Y 587.037,Z 443.678,A -85,B 0,C 180,E1 23459.605,E2 23459.605} C_VEL
LIN {X 0,Y 587.711,Z 213.286,A -85,B 0,C 180,E1 23456.394,E2 23456.394} C_VEL
LIN {X 0,Y 586.877,Z 208.332,A -85,B 0,C 180,E1 23456.243,E2 23456.243} C_VEL
LIN {X 0,Y 587.447,Z 157.447,A -85,B 0,C 180,E1 23452.964,E2 23452.964} C_VEL
LIN {X 0,Y 587.607,Z 137.976,A -85,B 0,C 180,E1 23451.668,E2 23451.668} C_VEL
LIN {X 0,Y 584.152,Z 129.665,A -85,B 0,C 180,E1 23450.802,E2 23450.802} C_VEL
LIN {X 0,Y 584.043,Z 129.279,A -85,B 0,C 180,E1 23450.189,E2 23450.189} C_VEL
LIN {X 0,Y 584.038,Z 129.285,A -85,B 0,C 180,E1 23447.26,E2 23447.26} C_VEL
LIN {X 0,Y 584.026,Z 129.29,A -85,B 0,C 180,E1 23444.026,E2 23444.026} C_VEL
LIN {X 0,Y 584.064,Z 129.296,A -85,B 0,C 180,E1 23440.97,E2 23440.97} C_VEL
LIN {X 0,Y 584.016,Z 129.296,A -85,B 0,C 180,E1 23437.887,E2 23437.887} C_VEL
LIN {X 0,Y 584.076,Z 129.288,A -85,B 0,C 180,E1 23434.873,E2 23434.873} C_VEL
LIN {X 0,Y 584.019,Z 129.291,A -85,B 0,C 180,E1 23431.824,E2 23431.824} C_VEL
LIN {X 0,Y 584.1,Z 129.293,A -85,B 0,C 180,E1 23428.752,E2 23428.752} C_VEL
LIN {X 0,Y 584.025,Z 129.288,A -85,B 0,C 180,E1 23425.667,E2 23425.667} C_VEL
LIN {X 0,Y 584.088,Z 129.291,A -85,B 0,C 180,E1 23422.548,E2 23422.548} C_VEL
LIN {X 0,Y 584.034,Z 129.288,A -85,B 0,C 180,E1 23419.502,E2 23419.502} C_VEL
LIN {X 0,Y 584.064,Z 129.291,A -85,B 0,C 180,E1 23416.305,E2 23416.305} C_VEL
LIN {X 0,Y 584.055,Z 129.292,A -85,B 0,C 180,E1 23413.262,E2 23413.262} C_VEL
LIN {X 0,Y 584.046,Z 129.29,A -85,B 0,C 180,E1 23409.957,E2 23409.957} C_VEL
LIN {X 0,Y 584.103,Z 129.292,A -85,B 0,C 180,E1 23406.877,E2 23406.877} C_VEL
LIN {X 0,Y 584.047,Z 129.29,A -85,B 0,C 180,E1 23403.632,E2 23403.632} C_VEL
LIN {X 0,Y 584.086,Z 129.286,A -85,B 0,C 180,E1 23400.392,E2 23400.392} C_VEL
LIN {X 0,Y 584.08,Z 129.294,A -85,B 0,C 180,E1 23397.155,E2 23397.155} C_VEL
LIN {X 0,Y 584.057,Z 129.289,A -85,B 0,C 180,E1 23393.907,E2 23393.907} C_VEL
LIN {X 0,Y 584.098,Z 129.288,A -85,B 0,C 180,E1 23390.74,E2 23390.74} C_VEL
LIN {X 0,Y 584.063,Z 129.291,A -85,B 0,C 180,E1 23387.544,E2 23387.544} C_VEL
LIN {X 0,Y 584.088,Z 129.28,A -85,B 0,C 180,E1 23384.308,E2 23384.308} C_VEL
LIN {X 0,Y 584.101,Z 129.292,A -85,B 0,C 180,E1 23381.02,E2 23381.02} C_VEL
LIN {X 0,Y 584.065,Z 129.283,A -85,B 0,C 180,E1 23377.77,E2 23377.77} C_VEL
LIN {X 0,Y 584.094,Z 129.285,A -85,B 0,C 180,E1 23374.554,E2 23374.554} C_VEL
LIN {X 0,Y 584.095,Z 129.289,A -85,B 0,C 180,E1 23371.213,E2 23371.213} C_VEL
LIN {X 0,Y 584.076,Z 129.283,A -85,B 0,C 180,E1 23367.924,E2 23367.924} C_VEL
LIN {X 0,Y 584.087,Z 129.288,A -85,B 0,C 180,E1 23364.738,E2 23364.738} C_VEL
LIN {X 0,Y 584.084,Z 129.291,A -85,B 0,C 180,E1 23361.457,E2 23361.457} C_VEL
LIN {X 0,Y 584.09,Z 129.286,A -85,B 0,C 180,E1 23358.117,E2 23358.117} C_VEL
LIN {X 0,Y 584.082,Z 129.288,A -85,B 0,C 180,E1 23354.851,E2 23354.851} C_VEL
LIN {X 0,Y 584.078,Z 129.244,A -85,B 0,C 180,E1 23351.62,E2 23351.62} C_VEL
LIN {X 0,Y 584.137,Z 129.561,A -85,B 0,C 180,E1 23351.286,E2 23351.286} C_VEL
LIN {X 0,Y 585.202,Z 132.446,A -85,B 0,C 180,E1 23350.958,E2 23350.958} C_VEL
LIN {X 0,Y 588.211,Z 138.885,A -85,B 0,C 180,E1 23350.289,E2 23350.289} C_VEL
LIN {X 0,Y 588.076,Z 162.115,A -85,B 0,C 180,E1 23348.856,E2 23348.856} C_VEL
LIN {X 0,Y 588.92,Z 167.665,A -85,B 0,C 180,E1 23348.704,E2 23348.704} C_VEL
LIN {X 0,Y 588.187,Z 375.191,A -85,B 0,C 180,E1 23345.645,E2 23345.645} C_VEL
LIN {X 0,Y 587.711,Z 510.624,A -85,B 0,C 180,E1 23343.676,E2 23343.676} C_VEL
LIN {X 0,Y 587.465,Z 534.326,A -85,B 0,C 180,E1 23343.146,E2 23343.146} C_VEL
LIN {X 0,Y 587.253,Z 554.822,A -85,B 0,C 180,E1 23342.523,E2 23342.523} C_VEL
LIN {X 0,Y 586.874,Z 578.144,A -85,B 0,C 180,E1 23341.617,E2 23341.617} C_VEL
LIN {X 0,Y 586.588,Z 599.565,A -85,B 0,C 180,E1 23340.595,E2 23340.595} C_VEL
LIN {X 0,Y 586.172,Z 620.051,A -85,B 0,C 180,E1 23339.422,E2 23339.422} C_VEL
LIN {X 0,Y 585.849,Z 640.337,A -85,B 0,C 180,E1 23338.073,E2 23338.073} C_VEL
LIN {X 0,Y 585.465,Z 658.931,A -85,B 0,C 180,E1 23336.634,E2 23336.634} C_VEL
LIN {X 0,Y 585.123,Z 678.126,A -85,B 0,C 180,E1 23334.933,E2 23334.933} C_VEL
LIN {X 0,Y 584.849,Z 695.175,A -85,B 0,C 180,E1 23333.207,E2 23333.207} C_VEL
LIN {X 0,Y 584.584,Z 710.996,A -85,B 0,C 180,E1 23331.364,E2 23331.364} C_VEL
LIN {X 0,Y 584.383,Z 725.917,A -85,B 0,C 180,E1 23329.385,E2 23329.385} C_VEL
LIN {X 0,Y 584.231,Z 738.74,A -85,B 0,C 180,E1 23327.427,E2 23327.427} C_VEL
LIN {X 0,Y 584.09,Z 750.796,A -85,B 0,C 180,E1 23325.285,E2 23325.285} C_VEL
LIN {X 0,Y 584.023,Z 760.542,A -85,B 0,C 180,E1 23323.262,E2 23323.262} C_VEL
LIN {X 0,Y 583.965,Z 769.339,A -85,B 0,C 180,E1 23321.055,E2 23321.055} C_VEL
LIN {X 0,Y 583.935,Z 776.174,A -85,B 0,C 180,E1 23318.964,E2 23318.964} C_VEL
LIN {X 0,Y 583.919,Z 781.841,A -85,B 0,C 180,E1 23316.686,E2 23316.686} C_VEL
LIN {X 0,Y 583.898,Z 785.594,A -85,B 0,C 180,E1 23314.616,E2 23314.616} C_VEL
LIN {X 0,Y 583.903,Z 788.055,A -85,B 0,C 180,E1 23312.355,E2 23312.355} C_VEL
LIN {X 0,Y 583.9,Z 788.939,A -85,B 0,C 180,E1 23310.294,E2 23310.294} C_VEL
LIN {X 0,Y 583.911,Z 788.323,A -85,B 0,C 180,E1 23308.037,E2 23308.037} C_VEL
LIN {X 0,Y 583.914,Z 786.39,A -85,B 0,C 180,E1 23305.974,E2 23305.974} C_VEL
LIN {X 0,Y 583.916,Z 782.461,A -85,B 0,C 180,E1 23303.61,E2 23303.61} C_VEL
LIN {X 0,Y 583.916,Z 777.805,A -85,B 0,C 180,E1 23301.631,E2 23301.631} C_VEL
LIN {X 0,Y 583.953,Z 770.763,A -85,B 0,C 180,E1 23299.344,E2 23299.344} C_VEL
LIN {X 0,Y 583.989,Z 763.107,A -85,B 0,C 180,E1 23297.341,E2 23297.341} C_VEL
LIN {X 0,Y 584.068,Z 752.881,A -85,B 0,C 180,E1 23295.121,E2 23295.121} C_VEL
LIN {X 0,Y 584.172,Z 742.398,A -85,B 0,C 180,E1 23293.187,E2 23293.187} C_VEL
LIN {X 0,Y 584.33,Z 729.437,A -85,B 0,C 180,E1 23291.128,E2 23291.128} C_VEL
LIN {X 0,Y 584.544,Z 715.221,A -85,B 0,C 180,E1 23289.159,E2 23289.159} C_VEL
LIN {X 0,Y 584.76,Z 699.412,A -85,B 0,C 180,E1 23287.268,E2 23287.268} C_VEL
LIN {X 0,Y 585.067,Z 681.474,A -85,B 0,C 180,E1 23285.39,E2 23285.39} C_VEL
LIN {X 0,Y 585.425,Z 663.256,A -85,B 0,C 180,E1 23283.722,E2 23283.722} C_VEL
LIN {X 0,Y 585.732,Z 644.345,A -85,B 0,C 180,E1 23282.225,E2 23282.225} C_VEL
LIN {X 0,Y 586.144,Z 622.72,A -85,B 0,C 180,E1 23280.745,E2 23280.745} C_VEL
LIN {X 0,Y 586.503,Z 602.855,A -85,B 0,C 180,E1 23279.582,E2 23279.582} C_VEL
LIN {X 0,Y 586.848,Z 581.244,A -85,B 0,C 180,E1 23278.521,E2 23278.521} C_VEL
LIN {X 0,Y 587.157,Z 560.545,A -85,B 0,C 180,E1 23277.677,E2 23277.677} C_VEL
LIN {X 0,Y 587.441,Z 537.907,A -85,B 0,C 180,E1 23276.953,E2 23276.953} C_VEL
LIN {X 0,Y 587.629,Z 516.816,A -85,B 0,C 180,E1 23276.44,E2 23276.44} C_VEL
LIN {X 0,Y 587.819,Z 485.751,A -85,B 0,C 180,E1 23275.942,E2 23275.942} C_VEL
LIN {X 0,Y 588.532,Z 274.541,A -85,B 0,C 180,E1 23272.885,E2 23272.885} C_VEL
LIN {X 0,Y 588.761,Z 165.644,A -85,B 0,C 180,E1 23271.253,E2 23271.253} C_VEL
LIN {X 0,Y 587.944,Z 160.547,A -85,B 0,C 180,E1 23271.071,E2 23271.071} C_VEL
LIN {X 0,Y 588.141,Z 138.513,A -85,B 0,C 180,E1 23269.682,E2 23269.682} C_VEL
LIN {X 0,Y 584.17,Z 129.751,A -85,B 0,C 180,E1 23268.75,E2 23268.75} C_VEL
LIN {X 0,Y 584.08,Z 129.243,A -85,B 0,C 180,E1 23268.424,E2 23268.424} C_VEL
LIN {X 0,Y 584.081,Z 129.289,A -85,B 0,C 180,E1 23265.269,E2 23265.269} C_VEL
LIN {X 0,Y 584.085,Z 129.287,A -85,B 0,C 180,E1 23262.015,E2 23262.015} C_VEL
LIN {X 0,Y 584.093,Z 129.292,A -85,B 0,C 180,E1 23258.668,E2 23258.668} C_VEL
LIN {X 0,Y 584.087,Z 129.287,A -85,B 0,C 180,E1 23255.352,E2 23255.352} C_VEL
LIN {X 0,Y 584.075,Z 129.284,A -85,B 0,C 180,E1 23252.167,E2 23252.167} C_VEL
LIN {X 0,Y 584.097,Z 129.291,A -85,B 0,C 180,E1 23248.864,E2 23248.864} C_VEL
LIN {X 0,Y 584.098,Z 129.284,A -85,B 0,C 180,E1 23245.555,E2 23245.555} C_VEL
LIN {X 0,Y 584.067,Z 129.283,A -85,B 0,C 180,E1 23242.336,E2 23242.336} C_VEL
LIN {X 0,Y 584.096,Z 129.29,A -85,B 0,C 180,E1 23239.084,E2 23239.084} C_VEL
LIN {X 0,Y 584.081,Z 129.28,A -85,B 0,C 180,E1 23235.794,E2 23235.794} C_VEL
LIN {X 0,Y 584.067,Z 129.292,A -85,B 0,C 180,E1 23232.557,E2 23232.557} C_VEL
LIN {X 0,Y 584.097,Z 129.287,A -85,B 0,C 180,E1 23229.359,E2 23229.359} C_VEL
LIN {X 0,Y 584.057,Z 129.289,A -85,B 0,C 180,E1 23226.191,E2 23226.191} C_VEL
LIN {X 0,Y 584.095,Z 129.293,A -85,B 0,C 180,E1 23222.944,E2 23222.944} C_VEL
LIN {X 0,Y 584.076,Z 129.286,A -85,B 0,C 180,E1 23219.706,E2 23219.706} C_VEL
LIN {X 0,Y 584.054,Z 129.29,A -85,B 0,C 180,E1 23216.467,E2 23216.467} C_VEL
LIN {X 0,Y 584.1,Z 129.29,A -85,B 0,C 180,E1 23213.315,E2 23213.315} C_VEL
LIN {X 0,Y 584.045,Z 129.29,A -85,B 0,C 180,E1 23210.143,E2 23210.143} C_VEL
LIN {X 0,Y 584.08,Z 129.293,A -85,B 0,C 180,E1 23206.91,E2 23206.91} C_VEL
LIN {X 0,Y 584.061,Z 129.292,A -85,B 0,C 180,E1 23206.719,E2 23206.719} C_VEL
LIN {X 0,Y 583.039,Z 129.418,A -85,B 0,C 180,E1 23205.963,E2 23205.963} C_VEL
LIN {X 0,Y 576.682,Z 130.211,A -85,B 0,C 180,E1 23203.842,E2 23203.842} C_VEL
LIN {X 0,Y 576.161,Z 130.28,A -85,B 0,C 180,E1 23203.291,E2 23203.291} C_VEL
LIN {X 0,Y 576.098,Z 130.274,A -85,B 0,C 180,E1 23200.113,E2 23200.113} C_VEL
LIN {X 0,Y 576.13,Z 130.281,A -85,B 0,C 180,E1 23196.893,E2 23196.893} C_VEL
LIN {X 0,Y 576.109,Z 130.274,A -85,B 0,C 180,E1 23193.798,E2 23193.798} C_VEL
LIN {X 0,Y 576.099,Z 130.28,A -85,B 0,C 180,E1 23190.583,E2 23190.583} C_VEL
LIN {X 0,Y 576.126,Z 130.278,A -85,B 0,C 180,E1 23187.57,E2 23187.57} C_VEL
LIN {X 0,Y 576.085,Z 130.275,A -85,B 0,C 180,E1 23184.449,E2 23184.449} C_VEL
LIN {X 0,Y 576.151,Z 130.283,A -85,B 0,C 180,E1 23181.336,E2 23181.336} C_VEL
LIN {X 0,Y 576.078,Z 130.285,A -85,B 0,C 180,E1 23178.204,E2 23178.204} C_VEL
LIN {X 0,Y 576.131,Z 130.281,A -85,B 0,C 180,E1 23175.062,E2 23175.062} C_VEL
LIN {X 0,Y 576.08,Z 130.274,A -85,B 0,C 180,E1 23172.025,E2 23172.025} C_VEL
LIN {X 0,Y 576.136,Z 130.518,A -85,B 0,C 180,E1 23169.722,E2 23169.722} C_VEL
LIN {X 0,Y 577.61,Z 134.007,A -85,B 0,C 180,E1 23169.306,E2 23169.306} C_VEL
LIN {X 0,Y 580.95,Z 142.167,A -85,B 0,C 180,E1 23168.473,E2 23168.473} C_VEL
LIN {X 0,Y 580.209,Z 187.046,A -85,B 0,C 180,E1 23165.502,E2 23165.502} C_VEL
LIN {X 0,Y 580.022,Z 209.367,A -85,B 0,C 180,E1 23164.081,E2 23164.081} C_VEL
LIN {X 0,Y 581.022,Z 216.047,A -85,B 0,C 180,E1 23163.915,E2 23163.915} C_VEL
LIN {X 0,Y 580.119,Z 447.044,A -85,B 0,C 180,E1 23160.658,E2 23160.658} C_VEL
LIN {X 0,Y 579.82,Z 515.779,A -85,B 0,C 180,E1 23159.677,E2 23159.677} C_VEL
LIN {X 0,Y 579.564,Z 537.03,A -85,B 0,C 180,E1 23159.186,E2 23159.186} C_VEL
LIN {X 0,Y 579.246,Z 558.983,A -85,B 0,C 180,E1 23158.491,E2 23158.491} C_VEL
LIN {X 0,Y 578.933,Z 579.585,A -85,B 0,C 180,E1 23157.652,E2 23157.652} C_VEL
LIN {X 0,Y 578.509,Z 599.443,A -85,B 0,C 180,E1 23156.647,E2 23156.647} C_VEL
LIN {X 0,Y 578.086,Z 619.993,A -85,B 0,C 180,E1 23155.4,E2 23155.4} C_VEL
LIN {X 0,Y 577.704,Z 638.743,A -85,B 0,C 180,E1 23154.053,E2 23154.053} C_VEL
LIN {X 0,Y 577.307,Z 656.503,A -85,B 0,C 180,E1 23152.558,E2 23152.558} C_VEL
LIN {X 0,Y 576.955,Z 672.764,A -85,B 0,C 180,E1 23150.968,E2 23150.968} C_VEL
LIN {X 0,Y 576.648,Z 689.009,A -85,B 0,C 180,E1 23149.129,E2 23149.129} C_VEL
LIN {X 0,Y 576.432,Z 702.529,A -85,B 0,C 180,E1 23147.358,E2 23147.358} C_VEL
LIN {X 0,Y 576.239,Z 714.694,A -85,B 0,C 180,E1 23145.498,E2 23145.498} C_VEL
LIN {X 0,Y 576.093,Z 726.085,A -85,B 0,C 180,E1 23143.448,E2 23143.448} C_VEL
LIN {X 0,Y 576.006,Z 735.572,A -85,B 0,C 180,E1 23141.413,E2 23141.413} C_VEL
LIN {X 0,Y 575.949,Z 743.227,A -85,B 0,C 180,E1 23139.392,E2 23139.392} C_VEL
LIN {X 0,Y 575.921,Z 749.531,A -85,B 0,C 180,E1 23137.281,E2 23137.281} C_VEL
LIN {X 0,Y 575.914,Z 754.243,A -85,B 0,C 180,E1 23135.179,E2 23135.179} C_VEL
LIN {X 0,Y 575.912,Z 757.233,A -85,B 0,C 180,E1 23133.085,E2 23133.085} C_VEL
LIN {X 0,Y 575.91,Z 758.796,A -85,B 0,C 180,E1 23130.895,E2 23130.895} C_VEL
LIN {X 0,Y 575.914,Z 758.749,A -85,B 0,C 180,E1 23128.806,E2 23128.806} C_VEL
LIN {X 0,Y 575.915,Z 757.015,A -85,B 0,C 180,E1 23126.631,E2 23126.631} C_VEL
LIN {X 0,Y 575.917,Z 753.608,A -85,B 0,C 180,E1 23124.421,E2 23124.421} C_VEL
LIN {X 0,Y 575.916,Z 748.997,A -85,B 0,C 180,E1 23122.418,E2 23122.418} C_VEL
LIN {X 0,Y 575.946,Z 742.479,A -85,B 0,C 180,E1 23120.306,E2 23120.306} C_VEL
LIN {X 0,Y 576.017,Z 734.483,A -85,B 0,C 180,E1 23118.238,E2 23118.238} C_VEL
LIN {X 0,Y 576.105,Z 724.983,A -85,B 0,C 180,E1 23116.245,E2 23116.245} C_VEL
LIN {X 0,Y 576.244,Z 713.33,A -85,B 0,C 180,E1 23114.192,E2 23114.192} C_VEL
LIN {X 0,Y 576.452,Z 700.945,A -85,B 0,C 180,E1 23112.33,E2 23112.33} C_VEL
LIN {X 0,Y 576.692,Z 687.184,A -85,B 0,C 180,E1 23110.557,E2 23110.557} C_VEL
LIN {X 0,Y 576.971,Z 672.104,A -85,B 0,C 180,E1 23108.873,E2 23108.873} C_VEL
LIN {X 0,Y 577.326,Z 655.101,A -85,B 0,C 180,E1 23107.228,E2 23107.228} C_VEL
LIN {X 0,Y 577.739,Z 637.133,A -85,B 0,C 180,E1 23105.731,E2 23105.731} C_VEL
LIN {X 0,Y 578.144,Z 618.087,A -85,B 0,C 180,E1 23104.384,E2 23104.384} C_VEL
LIN {X 0,Y 578.53,Z 598.078,A -85,B 0,C 180,E1 23103.188,E2 23103.188} C_VEL
LIN {X 0,Y 578.956,Z 577.253,A -85,B 0,C 180,E1 23102.157,E2 23102.157} C_VEL
LIN {X 0,Y 579.289,Z 557.24,A -85,B 0,C 180,E1 23101.355,E2 23101.355} C_VEL
LIN {X 0,Y 579.572,Z 535.719,A -85,B 0,C 180,E1 23100.689,E2 23100.689} C_VEL
LIN {X 0,Y 579.827,Z 514.263,A -85,B 0,C 180,E1 23100.208,E2 23100.208} C_VEL
LIN {X 0,Y 580.725,Z 286.24,A -85,B 0,C 180,E1 23096.995,E2 23096.995} C_VEL
LIN {X 0,Y 580.836,Z 213.722,A -85,B 0,C 180,E1 23095.949,E2 23095.949} C_VEL
LIN {X 0,Y 579.931,Z 208.142,A -85,B 0,C 180,E1 23095.773,E2 23095.773} C_VEL
LIN {X 0,Y 580.689,Z 158.24,A -85,B 0,C 180,E1 23092.514,E2 23092.514} C_VEL
LIN {X 0,Y 580.917,Z 141.53,A -85,B 0,C 180,E1 23091.39,E2 23091.39} C_VEL
LIN {X 0,Y 576.164,Z 130.649,A -85,B 0,C 180,E1 23090.219,E2 23090.219} C_VEL
LIN {X 0,Y 576.09,Z 130.286,A -85,B 0,C 180,E1 23089.481,E2 23089.481} C_VEL
LIN {X 0,Y 576.101,Z 130.287,A -85,B 0,C 180,E1 23086.174,E2 23086.174} C_VEL
LIN {X 0,Y 576.101,Z 130.278,A -85,B 0,C 180,E1 23083.204,E2 23083.204} C_VEL
LIN {X 0,Y 576.079,Z 130.279,A -85,B 0,C 180,E1 23079.955,E2 23079.955} C_VEL
LIN {X 0,Y 576.132,Z 130.282,A -85,B 0,C 180,E1 23076.904,E2 23076.904} C_VEL
LIN {X 0,Y 576.078,Z 130.284,A -85,B 0,C 180,E1 23073.739,E2 23073.739} C_VEL
LIN {X 0,Y 576.142,Z 130.276,A -85,B 0,C 180,E1 23070.563,E2 23070.563} C_VEL
LIN {X 0,Y 576.089,Z 130.283,A -85,B 0,C 180,E1 23067.495,E2 23067.495} C_VEL
LIN {X 0,Y 576.107,Z 130.279,A -85,B 0,C 180,E1 23064.179,E2 23064.179} C_VEL
LIN {X 0,Y 576.109,Z 130.283,A -85,B 0,C 180,E1 23061.258,E2 23061.258} C_VEL
LIN {X 0,Y 576.1,Z 130.277,A -85,B 0,C 180,E1 23057.995,E2 23057.995} C_VEL
LIN {X 0,Y 576.159,Z 130.281,A -85,B 0,C 180,E1 23054.854,E2 23054.854} C_VEL
LIN {X 0,Y 576.101,Z 130.281,A -85,B 0,C 180,E1 23051.716,E2 23051.716} C_VEL
LIN {X 0,Y 576.152,Z 130.277,A -85,B 0,C 180,E1 23048.483,E2 23048.483} C_VEL
LIN {X 0,Y 576.117,Z 130.282,A -85,B 0,C 180,E1 23045.378,E2 23045.378} C_VEL
LIN {X 0,Y 576.114,Z 130.279,A -85,B 0,C 180,E1 23041.989,E2 23041.989} C_VEL
LIN {X 0,Y 576.161,Z 130.281,A -85,B 0,C 180,E1 23038.807,E2 23038.807} C_VEL
LIN {X 0,Y 576.115,Z 130.279,A -85,B 0,C 180,E1 23035.621,E2 23035.621} C_VEL
LIN {X 0,Y 576.148,Z 130.275,A -85,B 0,C 180,E1 23032.321,E2 23032.321} C_VEL
LIN {X 0,Y 576.155,Z 130.281,A -85,B 0,C 180,E1 23028.995,E2 23028.995} C_VEL
LIN {X 0,Y 576.121,Z 130.275,A -85,B 0,C 180,E1 23025.733,E2 23025.733} C_VEL
LIN {X 0,Y 576.159,Z 130.275,A -85,B 0,C 180,E1 23022.425,E2 23022.425} C_VEL
LIN {X 0,Y 576.159,Z 130.272,A -85,B 0,C 180,E1 23019.054,E2 23019.054} C_VEL
LIN {X 0,Y 576.13,Z 130.278,A -85,B 0,C 180,E1 23015.822,E2 23015.822} C_VEL
LIN {X 0,Y 576.152,Z 130.271,A -85,B 0,C 180,E1 23012.621,E2 23012.621} C_VEL
LIN {X 0,Y 576.148,Z 130.283,A -85,B 0,C 180,E1 23009.322,E2 23009.322} C_VEL
LIN {X 0,Y 576.143,Z 130.276,A -85,B 0,C 180,E1 23006.027,E2 23006.027} C_VEL
LIN {X 0,Y 576.148,Z 130.276,A -85,B 0,C 180,E1 23002.8,E2 23002.8} C_VEL
LIN {X 0,Y 576.141,Z 130.277,A -85,B 0,C 180,E1 22999.626,E2 22999.626} C_VEL
LIN {X 0,Y 576.156,Z 130.271,A -85,B 0,C 180,E1 22996.316,E2 22996.316} C_VEL
LIN {X 0,Y 576.147,Z 130.269,A -85,B 0,C 180,E1 22993,E2 22993} C_VEL
LIN {X 0,Y 576.184,Z 130.544,A -85,B 0,C 180,E1 22991.919,E2 22991.919} C_VEL
LIN {X 0,Y 577.489,Z 133.779,A -85,B 0,C 180,E1 22991.537,E2 22991.537} C_VEL
LIN {X 0,Y 581.669,Z 142.703,A -85,B 0,C 180,E1 22990.587,E2 22990.587} C_VEL
LIN {X 0,Y 581.499,Z 162.115,A -85,B 0,C 180,E1 22989.38,E2 22989.38} C_VEL
LIN {X 0,Y 582.664,Z 169.319,A -85,B 0,C 180,E1 22989.173,E2 22989.173} C_VEL
LIN {X 0,Y 581.675,Z 376.594,A -85,B 0,C 180,E1 22986.085,E2 22986.085} C_VEL
LIN {X 0,Y 581.042,Z 510.731,A -85,B 0,C 180,E1 22984.113,E2 22984.113} C_VEL
LIN {X 0,Y 580.713,Z 534.512,A -85,B 0,C 180,E1 22983.577,E2 22983.577} C_VEL
LIN {X 0,Y 580.421,Z 555.622,A -85,B 0,C 180,E1 22982.927,E2 22982.927} C_VEL
LIN {X 0,Y 579.953,Z 577.431,A -85,B 0,C 180,E1 22982.072,E2 22982.072} C_VEL
LIN {X 0,Y 579.543,Z 598.687,A -85,B 0,C 180,E1 22981.053,E2 22981.053} C_VEL
LIN {X 0,Y 578.993,Z 620.054,A -85,B 0,C 180,E1 22979.824,E2 22979.824} C_VEL
LIN {X 0,Y 578.529,Z 640.762,A -85,B 0,C 180,E1 22978.427,E2 22978.427} C_VEL
LIN {X 0,Y 578.02,Z 659.595,A -85,B 0,C 180,E1 22976.949,E2 22976.949} C_VEL
LIN {X 0,Y 577.555,Z 678.912,A -85,B 0,C 180,E1 22975.205,E2 22975.205} C_VEL
LIN {X 0,Y 577.18,Z 695.974,A -85,B 0,C 180,E1 22973.447,E2 22973.447} C_VEL
LIN {X 0,Y 576.822,Z 711.849,A -85,B 0,C 180,E1 22971.56,E2 22971.56} C_VEL
LIN {X 0,Y 576.528,Z 727.336,A -85,B 0,C 180,E1 22969.449,E2 22969.449} C_VEL
LIN {X 0,Y 576.325,Z 740.646,A -85,B 0,C 180,E1 22967.361,E2 22967.361} C_VEL
LIN {X 0,Y 576.149,Z 752.175,A -85,B 0,C 180,E1 22965.228,E2 22965.228} C_VEL
LIN {X 0,Y 576.051,Z 762.29,A -85,B 0,C 180,E1 22963.04,E2 22963.04} C_VEL
LIN {X 0,Y 575.978,Z 770.052,A -85,B 0,C 180,E1 22961.008,E2 22961.008} C_VEL
LIN {X 0,Y 575.931,Z 777.04,A -85,B 0,C 180,E1 22958.787,E2 22958.787} C_VEL
LIN {X 0,Y 575.922,Z 782.047,A -85,B 0,C 180,E1 22956.68,E2 22956.68} C_VEL
LIN {X 0,Y 575.897,Z 785.913,A -85,B 0,C 180,E1 22954.481,E2 22954.481} C_VEL
LIN {X 0,Y 575.903,Z 788.122,A -85,B 0,C 180,E1 22952.288,E2 22952.288} C_VEL
LIN {X 0,Y 575.911,Z 788.984,A -85,B 0,C 180,E1 22950.099,E2 22950.099} C_VEL
LIN {X 0,Y 575.909,Z 788.256,A -85,B 0,C 180,E1 22947.911,E2 22947.911} C_VEL
LIN {X 0,Y 575.906,Z 786.277,A -85,B 0,C 180,E1 22945.819,E2 22945.819} C_VEL
LIN {X 0,Y 575.922,Z 782.461,A -85,B 0,C 180,E1 22943.521,E2 22943.521} C_VEL
LIN {X 0,Y 575.92,Z 777.806,A -85,B 0,C 180,E1 22941.514,E2 22941.514} C_VEL
LIN {X 0,Y 575.97,Z 770.764,A -85,B 0,C 180,E1 22939.194,E2 22939.194} C_VEL
LIN {X 0,Y 576.034,Z 763.108,A -85,B 0,C 180,E1 22937.163,E2 22937.163} C_VEL
LIN {X 0,Y 576.137,Z 752.882,A -85,B 0,C 180,E1 22934.912,E2 22934.912} C_VEL
LIN {X 0,Y 576.281,Z 742.338,A -85,B 0,C 180,E1 22932.939,E2 22932.939} C_VEL
LIN {X 0,Y 576.481,Z 729.463,A -85,B 0,C 180,E1 22930.865,E2 22930.865} C_VEL
LIN {X 0,Y 576.773,Z 715.109,A -85,B 0,C 180,E1 22928.85,E2 22928.85} C_VEL
LIN {X 0,Y 577.086,Z 699.227,A -85,B 0,C 180,E1 22926.927,E2 22926.927} C_VEL
LIN {X 0,Y 577.491,Z 681.124,A -85,B 0,C 180,E1 22925.011,E2 22925.011} C_VEL
LIN {X 0,Y 577.969,Z 662.902,A -85,B 0,C 180,E1 22923.326,E2 22923.326} C_VEL
LIN {X 0,Y 578.435,Z 643.693,A -85,B 0,C 180,E1 22921.793,E2 22921.793} C_VEL
LIN {X 0,Y 578.947,Z 622.135,A -85,B 0,C 180,E1 22920.307,E2 22920.307} C_VEL
LIN {X 0,Y 579.47,Z 601.847,A -85,B 0,C 180,E1 22919.115,E2 22919.115} C_VEL
LIN {X 0,Y 579.904,Z 579.653,A -85,B 0,C 180,E1 22918.027,E2 22918.027} C_VEL
LIN {X 0,Y 580.405,Z 557.281,A -85,B 0,C 180,E1 22917.129,E2 22917.129} C_VEL
LIN {X 0,Y 580.704,Z 535.446,A -85,B 0,C 180,E1 22916.449,E2 22916.449} C_VEL
LIN {X 0,Y 581.034,Z 512.445,A -85,B 0,C 180,E1 22915.916,E2 22915.916} C_VEL
LIN {X 0,Y 581.327,Z 454.195,A -85,B 0,C 180,E1 22915.044,E2 22915.044} C_VEL
LIN {X 0,Y 582.29,Z 244.522,A -85,B 0,C 180,E1 22911.96,E2 22911.96} C_VEL
LIN {X 0,Y 582.51,Z 167.336,A -85,B 0,C 180,E1 22910.784,E2 22910.784} C_VEL
LIN {X 0,Y 581.372,Z 160.635,A -85,B 0,C 180,E1 22910.552,E2 22910.552} C_VEL
LIN {X 0,Y 581.61,Z 142.201,A -85,B 0,C 180,E1 22909.375,E2 22909.375} C_VEL
LIN {X 0,Y 576.297,Z 131.107,A -85,B 0,C 180,E1 22908.173,E2 22908.173} C_VEL
LIN {X 0,Y 576.152,Z 130.275,A -85,B 0,C 180,E1 22907.945,E2 22907.945} C_VEL
LIN {X 0,Y 576.153,Z 130.268,A -85,B 0,C 180,E1 22904.643,E2 22904.643} C_VEL
LIN {X 0,Y 576.147,Z 130.277,A -85,B 0,C 180,E1 22901.391,E2 22901.391} C_VEL
LIN {X 0,Y 576.14,Z 130.276,A -85,B 0,C 180,E1 22898.157,E2 22898.157} C_VEL
LIN {X 0,Y 576.156,Z 130.283,A -85,B 0,C 180,E1 22894.816,E2 22894.816} C_VEL
LIN {X 0,Y 576.154,Z 130.27,A -85,B 0,C 180,E1 22891.49,E2 22891.49} C_VEL
LIN {X 0,Y 576.133,Z 130.273,A -85,B 0,C 180,E1 22888.28,E2 22888.28} C_VEL
LIN {X 0,Y 576.158,Z 130.281,A -85,B 0,C 180,E1 22884.942,E2 22884.942} C_VEL
LIN {X 0,Y 576.157,Z 130.266,A -85,B 0,C 180,E1 22881.543,E2 22881.543} C_VEL
LIN {X 0,Y 576.127,Z 130.279,A -85,B 0,C 180,E1 22878.308,E2 22878.308} C_VEL
LIN {X 0,Y 576.16,Z 130.271,A -85,B 0,C 180,E1 22874.985,E2 22874.985} C_VEL
LIN {X 0,Y 576.153,Z 130.275,A -85,B 0,C 180,E1 22871.613,E2 22871.613} C_VEL
LIN {X 0,Y 576.122,Z 130.279,A -85,B 0,C 180,E1 22868.382,E2 22868.382} C_VEL
LIN {X 0,Y 576.159,Z 130.28,A -85,B 0,C 180,E1 22865.177,E2 22865.177} C_VEL
LIN {X 0,Y 576.121,Z 130.278,A -85,B 0,C 180,E1 22861.989,E2 22861.989} C_VEL
LIN {X 0,Y 576.125,Z 130.282,A -85,B 0,C 180,E1 22858.608,E2 22858.608} C_VEL
LIN {X 0,Y 576.157,Z 130.275,A -85,B 0,C 180,E1 22855.421,E2 22855.421} C_VEL
LIN {X 0,Y 576.106,Z 130.279,A -85,B 0,C 180,E1 22852.22,E2 22852.22} C_VEL
LIN {X 0,Y 576.149,Z 130.281,A -85,B 0,C 180,E1 22848.995,E2 22848.995} C_VEL
LIN {X 0,Y 576.117,Z 130.278,A -85,B 0,C 180,E1 22845.835,E2 22845.835} C_VEL
LIN {X 0,Y 576.161,Z 130.28,A -85,B 0,C 180,E1 22843.291,E2 22843.291} C_VEL
LIN {X 0,Y 575.16,Z 130.411,A -85,B 0,C 180,E1 22842.525,E2 22842.525} C_VEL
LIN {X 0,Y 568.68,Z 131.197,A -85,B 0,C 180,E1 22840.375,E2 22840.375} C_VEL
LIN {X 0,Y 568.174,Z 131.26,A -85,B 0,C 180,E1 22839.815,E2 22839.815} C_VEL
LIN {X 0,Y 568.16,Z 131.268,A -85,B 0,C 180,E1 22836.468,E2 22836.468} C_VEL
LIN {X 0,Y 568.218,Z 131.261,A -85,B 0,C 180,E1 22833.339,E2 22833.339} C_VEL
LIN {X 0,Y 568.151,Z 131.267,A -85,B 0,C 180,E1 22830.13,E2 22830.13} C_VEL
LIN {X 0,Y 568.182,Z 131.273,A -85,B 0,C 180,E1 22826.889,E2 22826.889} C_VEL
LIN {X 0,Y 568.154,Z 131.261,A -85,B 0,C 180,E1 22823.875,E2 22823.875} C_VEL
LIN {X 0,Y 568.148,Z 131.267,A -85,B 0,C 180,E1 22820.557,E2 22820.557} C_VEL
LIN {X 0,Y 568.187,Z 131.275,A -85,B 0,C 180,E1 22817.488,E2 22817.488} C_VEL
LIN {X 0,Y 568.137,Z 131.277,A -85,B 0,C 180,E1 22814.319,E2 22814.319} C_VEL
LIN {X 0,Y 568.206,Z 131.268,A -85,B 0,C 180,E1 22811.137,E2 22811.137} C_VEL
LIN {X 0,Y 568.194,Z 131.642,A -85,B 0,C 180,E1 22810.289,E2 22810.289} C_VEL
LIN {X 0,Y 574.238,Z 145.457,A -85,B 0,C 180,E1 22808.778,E2 22808.778} C_VEL
LIN {X 0,Y 573.331,Z 189.746,A -85,B 0,C 180,E1 22805.812,E2 22805.812} C_VEL
LIN {X 0,Y 573.132,Z 209.495,A -85,B 0,C 180,E1 22804.547,E2 22804.547} C_VEL
LIN {X 0,Y 574.377,Z 217.432,A -85,B 0,C 180,E1 22804.342,E2 22804.342} C_VEL
LIN {X 0,Y 573.231,Z 448.494,A -85,B 0,C 180,E1 22801.047,E2 22801.047} C_VEL
LIN {X 0,Y 572.865,Z 515.819,A -85,B 0,C 180,E1 22800.074,E2 22800.074} C_VEL
LIN {X 0,Y 572.542,Z 537.098,A -85,B 0,C 180,E1 22799.578,E2 22799.578} C_VEL
LIN {X 0,Y 572.171,Z 558.469,A -85,B 0,C 180,E1 22798.897,E2 22798.897} C_VEL
LIN {X 0,Y 571.758,Z 578.913,A -85,B 0,C 180,E1 22798.06,E2 22798.06} C_VEL
LIN {X 0,Y 571.246,Z 598.466,A -85,B 0,C 180,E1 22797.069,E2 22797.069} C_VEL
LIN {X 0,Y 570.727,Z 618.989,A -85,B 0,C 180,E1 22795.821,E2 22795.821} C_VEL
LIN {X 0,Y 570.213,Z 638.081,A -85,B 0,C 180,E1 22794.444,E2 22794.444} C_VEL
LIN {X 0,Y 569.709,Z 655.909,A -85,B 0,C 180,E1 22792.93,E2 22792.93} C_VEL
LIN {X 0,Y 569.27,Z 672.589,A -85,B 0,C 180,E1 22791.284,E2 22791.284} C_VEL
LIN {X 0,Y 568.888,Z 688.165,A -85,B 0,C 180,E1 22789.507,E2 22789.507} C_VEL
LIN {X 0,Y 568.596,Z 701.819,A -85,B 0,C 180,E1 22787.71,E2 22787.71} C_VEL
LIN {X 0,Y 568.328,Z 714.697,A -85,B 0,C 180,E1 22785.719,E2 22785.719} C_VEL
LIN {X 0,Y 568.152,Z 725.649,A -85,B 0,C 180,E1 22783.728,E2 22783.728} C_VEL
LIN {X 0,Y 568.038,Z 735.167,A -85,B 0,C 180,E1 22781.678,E2 22781.678} C_VEL
LIN {X 0,Y 567.96,Z 742.875,A -85,B 0,C 180,E1 22779.627,E2 22779.627} C_VEL
LIN {X 0,Y 567.922,Z 749.533,A -85,B 0,C 180,E1 22777.384,E2 22777.384} C_VEL
LIN {X 0,Y 567.913,Z 754.245,A -85,B 0,C 180,E1 22775.253,E2 22775.253} C_VEL
LIN {X 0,Y 567.913,Z 757.234,A -85,B 0,C 180,E1 22773.129,E2 22773.129} C_VEL
LIN {X 0,Y 567.911,Z 758.796,A -85,B 0,C 180,E1 22770.908,E2 22770.908} C_VEL
LIN {X 0,Y 567.913,Z 758.748,A -85,B 0,C 180,E1 22768.789,E2 22768.789} C_VEL
LIN {X 0,Y 567.915,Z 757.043,A -85,B 0,C 180,E1 22766.609,E2 22766.609} C_VEL
LIN {X 0,Y 567.917,Z 753.813,A -85,B 0,C 180,E1 22764.443,E2 22764.443} C_VEL
LIN {X 0,Y 567.922,Z 749.196,A -85,B 0,C 180,E1 22762.391,E2 22762.391} C_VEL
LIN {X 0,Y 567.96,Z 742.832,A -85,B 0,C 180,E1 22760.27,E2 22760.27} C_VEL
LIN {X 0,Y 568.043,Z 735.116,A -85,B 0,C 180,E1 22758.219,E2 22758.219} C_VEL
LIN {X 0,Y 568.157,Z 725.501,A -85,B 0,C 180,E1 22756.153,E2 22756.153} C_VEL
LIN {X 0,Y 568.337,Z 713.968,A -85,B 0,C 180,E1 22754.071,E2 22754.071} C_VEL
LIN {X 0,Y 568.595,Z 701.708,A -85,B 0,C 180,E1 22752.184,E2 22752.184} C_VEL
LIN {X 0,Y 568.894,Z 688.03,A -85,B 0,C 180,E1 22750.386,E2 22750.386} C_VEL
LIN {X 0,Y 569.283,Z 672.098,A -85,B 0,C 180,E1 22748.573,E2 22748.573} C_VEL
LIN {X 0,Y 569.74,Z 654.638,A -85,B 0,C 180,E1 22746.866,E2 22746.866} C_VEL
LIN {X 0,Y 570.236,Z 637.131,A -85,B 0,C 180,E1 22745.391,E2 22745.391} C_VEL
LIN {X 0,Y 570.758,Z 618.073,A -85,B 0,C 180,E1 22744.028,E2 22744.028} C_VEL
LIN {X 0,Y 571.258,Z 598.069,A -85,B 0,C 180,E1 22742.819,E2 22742.819} C_VEL
LIN {X 0,Y 571.778,Z 577.118,A -85,B 0,C 180,E1 22741.771,E2 22741.771} C_VEL
LIN {X 0,Y 572.229,Z 556.478,A -85,B 0,C 180,E1 22740.939,E2 22740.939} C_VEL
LIN {X 0,Y 572.558,Z 535.045,A -85,B 0,C 180,E1 22740.276,E2 22740.276} C_VEL
LIN {X 0,Y 572.883,Z 512.821,A -85,B 0,C 180,E1 22739.786,E2 22739.786} C_VEL
LIN {X 0,Y 574.012,Z 285.885,A -85,B 0,C 180,E1 22736.554,E2 22736.554} C_VEL
LIN {X 0,Y 574.197,Z 215.238,A -85,B 0,C 180,E1 22735.524,E2 22735.524} C_VEL
LIN {X 0,Y 573.026,Z 208.129,A -85,B 0,C 180,E1 22735.302,E2 22735.302} C_VEL
LIN {X 0,Y 573.966,Z 159.053,A -85,B 0,C 180,E1 22732.054,E2 22732.054} C_VEL
LIN {X 0,Y 574.171,Z 145.293,A -85,B 0,C 180,E1 22731.115,E2 22731.115} C_VEL
LIN {X 0,Y 568.204,Z 131.651,A -85,B 0,C 180,E1 22729.624,E2 22729.624} C_VEL
LIN {X 0,Y 568.21,Z 131.269,A -85,B 0,C 180,E1 22728.845,E2 22728.845} C_VEL
LIN {X 0,Y 568.144,Z 131.276,A -85,B 0,C 180,E1 22725.681,E2 22725.681} C_VEL
LIN {X 0,Y 568.193,Z 131.274,A -85,B 0,C 180,E1 22722.498,E2 22722.498} C_VEL
LIN {X 0,Y 568.142,Z 131.267,A -85,B 0,C 180,E1 22719.443,E2 22719.443} C_VEL
LIN {X 0,Y 568.15,Z 131.261,A -85,B 0,C 180,E1 22716.124,E2 22716.124} C_VEL
LIN {X 0,Y 568.177,Z 131.274,A -85,B 0,C 180,E1 22713.061,E2 22713.061} C_VEL
LIN {X 0,Y 568.145,Z 131.268,A -85,B 0,C 180,E1 22709.82,E2 22709.82} C_VEL
LIN {X 0,Y 568.215,Z 131.262,A -85,B 0,C 180,E1 22706.636,E2 22706.636} C_VEL
LIN {X 0,Y 568.157,Z 131.269,A -85,B 0,C 180,E1 22703.436,E2 22703.436} C_VEL
LIN {X 0,Y 568.164,Z 131.261,A -85,B 0,C 180,E1 22700.07,E2 22700.07} C_VEL
LIN {X 0,Y 568.201,Z 131.268,A -85,B 0,C 180,E1 22696.984,E2 22696.984} C_VEL
LIN {X 0,Y 568.159,Z 131.268,A -85,B 0,C 180,E1 22693.744,E2 22693.744} C_VEL
LIN {X 0,Y 568.215,Z 131.267,A -85,B 0,C 180,E1 22690.545,E2 22690.545} C_VEL
LIN {X 0,Y 568.175,Z 131.27,A -85,B 0,C 180,E1 22687.381,E2 22687.381} C_VEL
LIN {X 0,Y 568.177,Z 131.265,A -85,B 0,C 180,E1 22684.037,E2 22684.037} C_VEL
LIN {X 0,Y 568.222,Z 131.267,A -85,B 0,C 180,E1 22680.807,E2 22680.807} C_VEL
LIN {X 0,Y 568.176,Z 131.27,A -85,B 0,C 180,E1 22677.58,E2 22677.58} C_VEL
LIN {X 0,Y 568.199,Z 131.265,A -85,B 0,C 180,E1 22674.244,E2 22674.244} C_VEL
LIN {X 0,Y 568.221,Z 131.27,A -85,B 0,C 180,E1 22670.99,E2 22670.99} C_VEL
LIN {X 0,Y 568.182,Z 131.268,A -85,B 0,C 180,E1 22667.706,E2 22667.706} C_VEL
LIN {X 0,Y 568.219,Z 131.255,A -85,B 0,C 180,E1 22664.487,E2 22664.487} C_VEL
LIN {X 0,Y 568.218,Z 131.272,A -85,B 0,C 180,E1 22661.109,E2 22661.109} C_VEL
LIN {X 0,Y 568.188,Z 131.257,A -85,B 0,C 180,E1 22657.769,E2 22657.769} C_VEL
LIN {X 0,Y 568.22,Z 131.261,A -85,B 0,C 180,E1 22654.462,E2 22654.462} C_VEL
LIN {X 0,Y 568.218,Z 131.268,A -85,B 0,C 180,E1 22651.06,E2 22651.06} C_VEL
LIN {X 0,Y 568.196,Z 131.26,A -85,B 0,C 180,E1 22647.779,E2 22647.779} C_VEL
LIN {X 0,Y 568.214,Z 131.262,A -85,B 0,C 180,E1 22644.502,E2 22644.502} C_VEL
LIN {X 0,Y 568.217,Z 131.27,A -85,B 0,C 180,E1 22641.083,E2 22641.083} C_VEL
LIN {X 0,Y 568.201,Z 131.268,A -85,B 0,C 180,E1 22637.763,E2 22637.763} C_VEL
LIN {X 0,Y 568.212,Z 131.264,A -85,B 0,C 180,E1 22634.453,E2 22634.453} C_VEL
LIN {X 0,Y 568.24,Z 131.501,A -85,B 0,C 180,E1 22632.575,E2 22632.575} C_VEL
LIN {X 0,Y 569.496,Z 134.673,A -85,B 0,C 180,E1 22632.192,E2 22632.192} C_VEL
LIN {X 0,Y 575.13,Z 146.299,A -85,B 0,C 180,E1 22630.908,E2 22630.908} C_VEL
LIN {X 0,Y 574.971,Z 162.115,A -85,B 0,C 180,E1 22629.916,E2 22629.916} C_VEL
LIN {X 0,Y 576.448,Z 170.93,A -85,B 0,C 180,E1 22629.653,E2 22629.653} C_VEL
LIN {X 0,Y 575.198,Z 378.109,A -85,B 0,C 180,E1 22626.533,E2 22626.533} C_VEL
LIN {X 0,Y 574.408,Z 510.839,A -85,B 0,C 180,E1 22624.561,E2 22624.561} C_VEL
LIN {X 0,Y 573.995,Z 534.666,A -85,B 0,C 180,E1 22624.019,E2 22624.019} C_VEL
LIN {X 0,Y 573.619,Z 556.217,A -85,B 0,C 180,E1 22623.347,E2 22623.347} C_VEL
LIN {X 0,Y 573.021,Z 578.707,A -85,B 0,C 180,E1 22622.448,E2 22622.448} C_VEL
LIN {X 0,Y 572.504,Z 599.805,A -85,B 0,C 180,E1 22621.42,E2 22621.42} C_VEL
LIN {X 0,Y 571.825,Z 620.948,A -85,B 0,C 180,E1 22620.178,E2 22620.178} C_VEL
LIN {X 0,Y 571.198,Z 642.117,A -85,B 0,C 180,E1 22618.72,E2 22618.72} C_VEL
LIN {X 0,Y 570.596,Z 660.259,A -85,B 0,C 180,E1 22617.272,E2 22617.272} C_VEL
LIN {X 0,Y 570.012,Z 679.465,A -85,B 0,C 180,E1 22615.507,E2 22615.507} C_VEL
LIN {X 0,Y 569.516,Z 696.623,A -85,B 0,C 180,E1 22613.705,E2 22613.705} C_VEL
LIN {X 0,Y 569.066,Z 712.698,A -85,B 0,C 180,E1 22611.76,E2 22611.76} C_VEL
LIN {X 0,Y 568.715,Z 727.338,A -85,B 0,C 180,E1 22609.727,E2 22609.727} C_VEL
LIN {X 0,Y 568.448,Z 740.012,A -85,B 0,C 180,E1 22607.715,E2 22607.715} C_VEL
LIN {X 0,Y 568.221,Z 751.32,A -85,B 0,C 180,E1 22605.618,E2 22605.618} C_VEL
LIN {X 0,Y 568.096,Z 761.457,A -85,B 0,C 180,E1 22603.433,E2 22603.433} C_VEL
LIN {X 0,Y 568.004,Z 769.697,A -85,B 0,C 180,E1 22601.267,E2 22601.267} C_VEL
LIN {X 0,Y 567.953,Z 776.776,A -85,B 0,C 180,E1 22599.014,E2 22599.014} C_VEL
LIN {X 0,Y 567.925,Z 782.048,A -85,B 0,C 180,E1 22596.774,E2 22596.774} C_VEL
LIN {X 0,Y 567.898,Z 785.913,A -85,B 0,C 180,E1 22594.544,E2 22594.544} C_VEL
LIN {X 0,Y 567.903,Z 788.122,A -85,B 0,C 180,E1 22592.321,E2 22592.321} C_VEL
LIN {X 0,Y 567.91,Z 788.984,A -85,B 0,C 180,E1 22590.101,E2 22590.101} C_VEL
LIN {X 0,Y 567.908,Z 788.256,A -85,B 0,C 180,E1 22587.881,E2 22587.881} C_VEL
LIN {X 0,Y 567.903,Z 786.277,A -85,B 0,C 180,E1 22585.759,E2 22585.759} C_VEL
LIN {X 0,Y 567.925,Z 782.461,A -85,B 0,C 180,E1 22583.429,E2 22583.429} C_VEL
LIN {X 0,Y 567.929,Z 777.806,A -85,B 0,C 180,E1 22581.394,E2 22581.394} C_VEL
LIN {X 0,Y 567.991,Z 770.765,A -85,B 0,C 180,E1 22579.041,E2 22579.041} C_VEL
LIN {X 0,Y 568.077,Z 763.109,A -85,B 0,C 180,E1 22576.98,E2 22576.98} C_VEL
LIN {X 0,Y 568.21,Z 752.617,A -85,B 0,C 180,E1 22574.642,E2 22574.642} C_VEL
LIN {X 0,Y 568.414,Z 741.821,A -85,B 0,C 180,E1 22572.601,E2 22572.601} C_VEL
LIN {X 0,Y 568.679,Z 728.578,A -85,B 0,C 180,E1 22570.458,E2 22570.458} C_VEL
LIN {X 0,Y 569.03,Z 714.388,A -85,B 0,C 180,E1 22568.455,E2 22568.455} C_VEL
LIN {X 0,Y 569.433,Z 698.968,A -85,B 0,C 180,E1 22566.568,E2 22566.568} C_VEL
LIN {X 0,Y 569.951,Z 681.124,A -85,B 0,C 180,E1 22564.657,E2 22564.657} C_VEL
LIN {X 0,Y 570.536,Z 662.903,A -85,B 0,C 180,E1 22562.951,E2 22562.951} C_VEL
LIN {X 0,Y 571.144,Z 643.622,A -85,B 0,C 180,E1 22561.394,E2 22561.394} C_VEL
LIN {X 0,Y 571.764,Z 622.728,A -85,B 0,C 180,E1 22559.934,E2 22559.934} C_VEL
LIN {X 0,Y 572.4,Z 602.849,A -85,B 0,C 180,E1 22558.75,E2 22558.75} C_VEL
LIN {X 0,Y 572.973,Z 580.423,A -85,B 0,C 180,E1 22557.629,E2 22557.629} C_VEL
LIN {X 0,Y 573.584,Z 558.394,A -85,B 0,C 180,E1 22556.729,E2 22556.729} C_VEL
LIN {X 0,Y 573.979,Z 536.114,A -85,B 0,C 180,E1 22556.022,E2 22556.022} C_VEL
LIN {X 0,Y 574.393,Z 513.301,A -85,B 0,C 180,E1 22555.482,E2 22555.482} C_VEL
LIN {X 0,Y 574.729,Z 461.7,A -85,B 0,C 180,E1 22554.696,E2 22554.696} C_VEL
LIN {X 0,Y 575.949,Z 250.951,A -85,B 0,C 180,E1 22551.565,E2 22551.565} C_VEL
LIN {X 0,Y 576.288,Z 168.971,A -85,B 0,C 180,E1 22550.303,E2 22550.303} C_VEL
LIN {X 0,Y 574.85,Z 160.547,A -85,B 0,C 180,E1 22550.009,E2 22550.009} C_VEL
LIN {X 0,Y 575.001,Z 146.061,A -85,B 0,C 180,E1 22549.065,E2 22549.065} C_VEL
LIN {X 0,Y 569.497,Z 134.671,A -85,B 0,C 180,E1 22547.808,E2 22547.808} C_VEL
LIN {X 0,Y 568.239,Z 131.501,A -85,B 0,C 180,E1 22547.425,E2 22547.425} C_VEL
LIN {X 0,Y 568.202,Z 131.256,A -85,B 0,C 180,E1 22544.261,E2 22544.261} C_VEL
LIN {X 0,Y 568.211,Z 131.261,A -85,B 0,C 180,E1 22540.986,E2 22540.986} C_VEL
LIN {X 0,Y 568.22,Z 131.262,A -85,B 0,C 180,E1 22537.632,E2 22537.632} C_VEL
LIN {X 0,Y 568.2,Z 131.268,A -85,B 0,C 180,E1 22534.384,E2 22534.384} C_VEL
LIN {X 0,Y 568.211,Z 131.262,A -85,B 0,C 180,E1 22531.154,E2 22531.154} C_VEL
LIN {X 0,Y 568.203,Z 131.258,A -85,B 0,C 180,E1 22527.909,E2 22527.909} C_VEL
LIN {X 0,Y 568.199,Z 131.27,A -85,B 0,C 180,E1 22524.531,E2 22524.531} C_VEL
LIN {X 0,Y 568.214,Z 131.256,A -85,B 0,C 180,E1 22521.253,E2 22521.253} C_VEL
LIN {X 0,Y 568.192,Z 131.266,A -85,B 0,C 180,E1 22518.042,E2 22518.042} C_VEL
LIN {X 0,Y 568.201,Z 131.262,A -85,B 0,C 180,E1 22514.678,E2 22514.678} C_VEL
LIN {X 0,Y 568.22,Z 131.266,A -85,B 0,C 180,E1 22511.366,E2 22511.366} C_VEL
LIN {X 0,Y 568.183,Z 131.267,A -85,B 0,C 180,E1 22508.093,E2 22508.093} C_VEL
LIN {X 0,Y 568.199,Z 131.27,A -85,B 0,C 180,E1 22504.744,E2 22504.744} C_VEL
LIN {X 0,Y 568.218,Z 131.265,A -85,B 0,C 180,E1 22501.512,E2 22501.512} C_VEL
LIN {X 0,Y 568.174,Z 131.269,A -85,B 0,C 180,E1 22498.286,E2 22498.286} C_VEL
LIN {X 0,Y 568.218,Z 131.27,A -85,B 0,C 180,E1 22495.054,E2 22495.054} C_VEL
LIN {X 0,Y 568.178,Z 131.266,A -85,B 0,C 180,E1 22491.907,E2 22491.907} C_VEL
LIN {X 0,Y 568.173,Z 131.27,A -85,B 0,C 180,E1 22488.53,E2 22488.53} C_VEL
LIN {X 0,Y 568.224,Z 131.266,A -85,B 0,C 180,E1 22485.322,E2 22485.322} C_VEL
LIN {X 0,Y 568.161,Z 131.265,A -85,B 0,C 180,E1 22482.169,E2 22482.169} C_VEL
LIN {X 0,Y 568.174,Z 131.26,A -85,B 0,C 180,E1 22479.815,E2 22479.815} C_VEL
LIN {X 0,Y 567.222,Z 131.392,A -85,B 0,C 180,E1 22479.038,E2 22479.038} C_VEL
LIN {X 0,Y 560.666,Z 132.208,A -85,B 0,C 180,E1 22476.801,E2 22476.801} C_VEL
LIN {X 0,Y 560.217,Z 132.257,A -85,B 0,C 180,E1 22476.289,E2 22476.289} C_VEL
LIN {X 0,Y 560.265,Z 132.256,A -85,B 0,C 180,E1 22473.045,E2 22473.045} C_VEL
LIN {X 0,Y 560.221,Z 132.256,A -85,B 0,C 180,E1 22469.899,E2 22469.899} C_VEL
LIN {X 0,Y 560.215,Z 132.262,A -85,B 0,C 180,E1 22466.53,E2 22466.53} C_VEL
LIN {X 0,Y 560.275,Z 132.248,A -85,B 0,C 180,E1 22463.285,E2 22463.285} C_VEL
LIN {X 0,Y 560.203,Z 132.254,A -85,B 0,C 180,E1 22460.125,E2 22460.125} C_VEL
LIN {X 0,Y 560.231,Z 132.254,A -85,B 0,C 180,E1 22456.878,E2 22456.878} C_VEL
LIN {X 0,Y 560.213,Z 132.266,A -85,B 0,C 180,E1 22453.826,E2 22453.826} C_VEL
LIN {X 0,Y 560.268,Z 132.421,A -85,B 0,C 180,E1 22450.984,E2 22450.984} C_VEL
LIN {X 0,Y 560.713,Z 134.2,A -85,B 0,C 180,E1 22450.724,E2 22450.724} C_VEL
LIN {X 0,Y 567.312,Z 148.603,A -85,B 0,C 180,E1 22449.119,E2 22449.119} C_VEL
LIN {X 0,Y 567.445,Z 153.182,A -85,B 0,C 180,E1 22448.784,E2 22448.784} C_VEL
LIN {X 0,Y 566.329,Z 199.893,A -85,B 0,C 180,E1 22445.634,E2 22445.634} C_VEL
LIN {X 0,Y 566.269,Z 209.546,A -85,B 0,C 180,E1 22445.026,E2 22445.026} C_VEL
LIN {X 0,Y 567.763,Z 218.996,A -85,B 0,C 180,E1 22444.776,E2 22444.776} C_VEL
LIN {X 0,Y 566.372,Z 449.792,A -85,B 0,C 180,E1 22441.447,E2 22441.447} C_VEL
LIN {X 0,Y 565.939,Z 515.859,A -85,B 0,C 180,E1 22440.481,E2 22440.481} C_VEL
LIN {X 0,Y 565.546,Z 537.326,A -85,B 0,C 180,E1 22439.976,E2 22439.976} C_VEL
LIN {X 0,Y 565.093,Z 559.021,A -85,B 0,C 180,E1 22439.273,E2 22439.273} C_VEL
LIN {X 0,Y 564.596,Z 578.932,A -85,B 0,C 180,E1 22438.448,E2 22438.448} C_VEL
